VAR_INPUT
	id: INT;
END_VAR
CASE ID OF 
	1: 		GetMBMUData.s_Name:= 'Status';
			GetMBMUData.s_Type:= 'status';
			GetMBMUData.s_unit:= TO_STRING(data.e_BMS_Status);
	2: 		GetMBMUData.s_Name:= 'Power-on status';
			GetMBMUData.s_Type:= 'status';
			GetMBMUData.s_unit:= TO_STRING(data.e_BMS_PowerOnStatus);
	3:		GetMBMUData.s_Name:= 'Voltage';
			GetMBMUData.s_Type:= 'power';
			GetMBMUData.s_Unit:= 'VDC';
			GetMBMUData.i_precision:= 1;
			GetMBMUData.r_Data:= data.r_SystemVoltage;
	4:		GetMBMUData.s_Name:= 'Current';
			GetMBMUData.s_Type:= 'power';
			GetMBMUData.s_Unit:= 'A';
			GetMBMUData.i_precision:= 1;
			GetMBMUData.r_Data:= data.r_SystemCurrent;
	5:		GetMBMUData.s_Name:= 'Power';
			GetMBMUData.s_Type:= 'power';
			GetMBMUData.s_Unit:= 'kW';
			GetMBMUData.i_precision:= 1;
			GetMBMUData.r_Data:= data.r_SystemPower;
	6:		GetMBMUData.s_Name:= 'Max charge current';
			GetMBMUData.s_Type:= 'limit';
			GetMBMUData.s_Unit:= 'A';
			GetMBMUData.i_precision:= 1;
			GetMBMUData.r_Data:= data.r_MaxChargeCurrentAllowed;
	7:		GetMBMUData.s_Name:= 'Max discharge current';
			GetMBMUData.s_Type:= 'limit';
			GetMBMUData.s_Unit:= 'A';
			GetMBMUData.i_precision:= 1;
			GetMBMUData.r_Data:= data.r_MaxDischargeCurrentAllowed;
	8:		GetMBMUData.s_Name:= 'Max charge power';
			GetMBMUData.s_Type:= 'limit';
			GetMBMUData.s_Unit:= 'kW';
			GetMBMUData.i_precision:= 1;
			GetMBMUData.r_Data:= data.r_MaxChargePowerAllowed;
	9: 		GetMBMUData.s_Name:= 'Max discharge power';
			GetMBMUData.s_Type:= 'limit';
			GetMBMUData.s_Unit:= 'kW';
			GetMBMUData.i_precision:= 1;
			GetMBMUData.r_Data:= data.r_MaxDischargePowerAllowed;
	10:		GetMBMUData.s_Name:= 'Charge SOE';
			GetMBMUData.s_Type:= 'energy';
			GetMBMUData.s_Unit:= '%';
			GetMBMUData.i_precision:= 0;
			GetMBMUData.r_Data:= data.r_ChargeSOE;
	11:		GetMBMUData.s_Name:= 'Discharge SOE';                       
			GetMBMUData.s_Type:= 'energy';                       
			GetMBMUData.s_Unit:= '%';                               
			GetMBMUData.i_precision:= 0;                              
			GetMBMUData.r_Data:= data.r_DischargeSOE;
//	12:		GetMBMUData.s_Name:= 'Total charge energy';                       
//			GetMBMUData.s_Type:= 'energy';                       
//			GetMBMUData.s_Unit:= 'kWh';                               
//			GetMBMUData.i_precision:= 0;                              
//			GetMBMUData.r_Data:= data.r_HistAccChargeEnergy;
//	13:		GetMBMUData.s_Name:= 'Total discharge energy';                         
//			GetMBMUData.s_Type:= 'energy';                                 
//			GetMBMUData.s_Unit:= 'kWh';                                         
//			GetMBMUData.i_precision:= 0;                                        
//			GetMBMUData.r_Data:= data.r_HistAccDischargeEnergy;
			
	14:		GetMBMUData.s_Name:= 'Remaining charge energy';                         
			GetMBMUData.s_Type:= 'energy';                                 
			GetMBMUData.s_Unit:= 'kWh';                                         
			GetMBMUData.i_precision:= 0;                                        
			GetMBMUData.r_Data:= data.r_RemainingChargeEnergy;
	15:		GetMBMUData.s_Name:= 'Remaining discharge energy';                         
			GetMBMUData.s_Type:= 'energy';                                 
			GetMBMUData.s_Unit:= 'kWh';                                         
			GetMBMUData.i_precision:= 0;                                        
			GetMBMUData.r_Data:= data.r_RemainingDischargeEnergy;	
	16:		GetMBMUData.s_Name:= 'Max allowed voltage';                         
			GetMBMUData.s_Type:= 'limit';                                 
			GetMBMUData.s_Unit:= 'VDC';                                         
			GetMBMUData.i_precision:= 1;                                        
			GetMBMUData.r_Data:= data.r_MaxSystemVoltageAllowed;	
	17:		GetMBMUData.s_Name:= 'Min allowed voltage';                                     
			GetMBMUData.s_Type:= 'limit';                                     
			GetMBMUData.s_Unit:= 'VDC';                                             
			GetMBMUData.i_precision:= 1;                                            
			GetMBMUData.r_Data:= data.r_MinSystemVoltageAllowed;
			GetMBMUData.s_Type:= 'cell';                                        
			GetMBMUData.s_Unit:= 'VDC';                                                
			GetMBMUData.i_precision:= 2;                                               
			GetMBMUData.r_Data:= data.ar_CellVoltage[2];
	18:		GetMBMUData.s_Name:= 'SOH';
			GetMBMUData.s_Type:= 'status';
			GetMBMUData.s_Unit:= '%';
			GetMBMUData.i_precision:= 1;
			GetMBMUData.r_Data:= data.r_SOH;	
	19:		GetMBMUData.s_Name:= 'SOC actual';                          
			GetMBMUData.s_Type:= 'status';                  
			GetMBMUData.s_Unit:= '%';                            
			GetMBMUData.i_precision:= 1;                         
			GetMBMUData.r_Data:= data.r_SOC;
	20:		GetMBMUData.s_Name:= 'Cycle count';                          
			GetMBMUData.s_Type:= 'status';                                          
			GetMBMUData.s_unit:= TO_STRING(data.ui_CycleCount);
	ELSE	
		RETURN;			
END_CASE
END_METHOD

METHOD GetPowerModuleArrayData : ST_HMI_Monitor_ArrayDataFormat
VAR_IN_OUT CONSTANT
	data		: ST_Powermodule_get;
END_VAR

VAR_INPUT
	id: INT;
END_VAR
CASE ID OF 
	1: 		GetPowerModuleArrayData.s_Name:= 'Status';                                                
			GetPowerModuleArrayData.s_Type:= 'Status';                                                
			GetPowerModuleArrayData.s_Unit:= TO_STRING(data.e_Status);				                            
	2: 		GetPowerModuleArrayData.s_Name:= 'Inverter Mode';                                         
			GetPowerModuleArrayData.s_Type:= 'Status';                                                
			GetPowerModuleArrayData.s_Unit:= TO_STRING(data.e_InverterMode);					                     
	3:		GetPowerModuleArrayData.s_Name:= 'Power Mode';                                            
			GetPowerModuleArrayData.s_Type:= 'Status';                                                
			GetPowerModuleArrayData.s_Unit:= TO_STRING(data.e_PowerMode);						                       
	4:		GetPowerModuleArrayData.s_Name:= 'Fan state';                                             
			GetPowerModuleArrayData.s_Type:= 'Status';                                                
			GetPowerModuleArrayData.s_Unit:= SEL(data.b_FanFb,'OFF', 'RUNNING');						                
	5:		GetPowerModuleArrayData.s_Name:= 'MCCB state';                                            
			GetPowerModuleArrayData.s_Type:= 'Status';                                                
			GetPowerModuleArrayData.s_Unit:= SEL(data.b_MccbFb,'OPEN', 'CLOSED');						               
	6:		GetPowerModuleArrayData.s_Name:= 'MCCB tripstate';                                        
			GetPowerModuleArrayData.s_Type:= 'Status';                                                
			GetPowerModuleArrayData.s_Unit:= SEL(data.b_MccbTripOK,'TRIPPED', 'OK');						              
	7:		GetPowerModuleArrayData.s_Name:= 'D7 measurements OK';                                    
			GetPowerModuleArrayData.s_Type:= 'Ugrid statusword';                                      
			GetPowerModuleArrayData.s_Unit:= TO_STRING(data.UgridStatusWord.b_D7MeasurementsOK);						
	8:		GetPowerModuleArrayData.s_Name:= 'Synchronized to D7';                                    
			GetPowerModuleArrayData.s_Type:= 'Ugrid statusword';                                      
			GetPowerModuleArrayData.s_Unit:= TO_STRING(data.UgridStatusWord.b_SynchronizedToD7);      
	9: 		GetPowerModuleArrayData.s_Name:= 'Ready to DCcharge';                                     
			GetPowerModuleArrayData.s_Type:= 'statusword';                                            
			GetPowerModuleArrayData.s_Unit:= TO_STRING(data.StatusWord.b_ReadyToDCCharge);            
	10:		GetPowerModuleArrayData.s_Name:= 'Ready to operate';                                      
			GetPowerModuleArrayData.s_Type:= 'statusword';                                            
			GetPowerModuleArrayData.s_Unit:= TO_STRING(data.StatusWord.b_ReadyToOperate);
	11:		GetPowerModuleArrayData.s_Name:= 'Run enabled';                                           
			GetPowerModuleArrayData.s_Type:= 'statusword';                                            
			GetPowerModuleArrayData.s_Unit:= TO_STRING(data.StatusWord.b_RunEnabled);                 
	12:		GetPowerModuleArrayData.s_Name:= 'Running';                                               
			GetPowerModuleArrayData.s_Type:= 'statusword';                                            
			GetPowerModuleArrayData.s_Unit:= TO_STRING(data.StatusWord.b_Running);                    
	13:		GetPowerModuleArrayData.s_Name:= 'DC at reference';                                       
			GetPowerModuleArrayData.s_Type:= 'statusword';                                            
			GetPowerModuleArrayData.s_Unit:= TO_STRING(data.StatusWord.b_DCAtReference);              
	14:		GetPowerModuleArrayData.s_Name:= 'DC above limit';                                        
			GetPowerModuleArrayData.s_Type:= 'statusword';                                            
			GetPowerModuleArrayData.s_Unit:= TO_STRING(data.StatusWord.b_DCAboveLimit);               
	15:		GetPowerModuleArrayData.s_Name:= 'Quickstop active';                                      
			GetPowerModuleArrayData.s_Type:= 'statusword';                                            
			GetPowerModuleArrayData.s_Unit:= TO_STRING(NOT(data.StatusWord.b_QuickstopNotActive));    
	16:		GetPowerModuleArrayData.s_Name:= 'Warning';                                               
			GetPowerModuleArrayData.s_Type:= 'statusword';                                            
			GetPowerModuleArrayData.s_Unit:= TO_STRING(data.StatusWord.b_Warning);                    
	17:		GetPowerModuleArrayData.s_Name:= 'Fault';                                                 
			GetPowerModuleArrayData.s_Type:= 'statusword';                                            
			GetPowerModuleArrayData.s_Unit:= TO_STRING(data.StatusWord.b_Fault);                      
	18:		GetPowerModuleArrayData.s_Name:= 'MCCB control OK';                                       
			GetPowerModuleArrayData.s_Type:= 'statusword';                                            
			GetPowerModuleArrayData.s_Unit:= TO_STRING(NOT(data.StatusWord.b_MCCBControlNotOK));						
	19:		GetPowerModuleArrayData.s_Name:= 'Load';                                                   
			GetPowerModuleArrayData.s_Type:= 'AC';                                                    
			GetPowerModuleArrayData.s_Unit:= '%';                                                     
			GetPowerModuleArrayData.r_Data:= data.r_LoadPercent;                                      
			GetPowerModuleArrayData.i_precision := 1;	                                                
	20:		GetPowerModuleArrayData.s_Name:= 'Apparent Power';                                        
			GetPowerModuleArrayData.s_Type:= 'AC';                                                    
			GetPowerModuleArrayData.s_Unit:= 'kVA';                                                   
			GetPowerModuleArrayData.r_Data:= data.r_ApparentPower;                                    
			GetPowerModuleArrayData.i_precision := 0;                                                 
	21:		GetPowerModuleArrayData.s_Name:= 'Active Power';                                          
			GetPowerModuleArrayData.s_Type:= 'AC';                                                    
			GetPowerModuleArrayData.s_Unit:= 'kW';                                                    
			GetPowerModuleArrayData.r_Data:= data.r_ActivePower;                                      
			GetPowerModuleArrayData.i_precision := 1;                                                 
	22:		GetPowerModuleArrayData.s_Name:= 'Reactive Power';                                        
			GetPowerModuleArrayData.s_Type:= 'AC';                                                    
			GetPowerModuleArrayData.s_Unit:= 'kvar';                                                  
			GetPowerModuleArrayData.r_Data:= data.r_ReactivePower;                                    
			GetPowerModuleArrayData.i_precision := 1;                                                 
	23:		GetPowerModuleArrayData.s_Name:= 'Current';                                               
			GetPowerModuleArrayData.s_Type:= 'AC';                                                    
			GetPowerModuleArrayData.s_Unit:= 'A';                                                     
			GetPowerModuleArrayData.r_Data:= data.r_ACCurrent;                                        
			GetPowerModuleArrayData.i_precision := 1;                                                 
	24:		GetPowerModuleArrayData.s_Name:= 'Reactive Current';                                      
			GetPowerModuleArrayData.s_Type:= 'AC';                                                    
			GetPowerModuleArrayData.s_Unit:= 'A';                                                     
			GetPowerModuleArrayData.r_Data:= data.r_ReactiveCurrent;                                  
			GetPowerModuleArrayData.i_precision := 1;                                                 
	25:		GetPowerModuleArrayData.s_Name:= 'Active Current';                                        
			GetPowerModuleArrayData.s_Type:= 'AC';                                                    
			GetPowerModuleArrayData.s_Unit:= 'A';                                                     
			GetPowerModuleArrayData.r_Data:= data.r_ActiveCurrent;                                    
			GetPowerModuleArrayData.i_precision := 1;                                                 
	26:		GetPowerModuleArrayData.s_Name:= 'Supply Voltage';                                        
			GetPowerModuleArrayData.s_Type:= 'AC';                                                    
			GetPowerModuleArrayData.s_Unit:= 'VAC';                                                   
			GetPowerModuleArrayData.r_Data:= data.r_ACVoltageSupply;                                  
			GetPowerModuleArrayData.i_precision := 1;                                                 
	27:		GetPowerModuleArrayData.s_Name:= 'Supply Frequency';                                      
			GetPowerModuleArrayData.s_Type:= 'AC';                                                    
			GetPowerModuleArrayData.s_Unit:= 'Hz';                                                    
			GetPowerModuleArrayData.r_Data:= data.r_FrequencySupply;                                  
			GetPowerModuleArrayData.i_precision := 2;                                                 
	28:		GetPowerModuleArrayData.s_Name:= 'Current';                                               
			GetPowerModuleArrayData.s_Type:= 'DC';                                                    
			GetPowerModuleArrayData.s_Unit:= 'A';                                                     
			GetPowerModuleArrayData.r_Data:= data.r_DCCurrent;                                        
			GetPowerModuleArrayData.i_precision := 1;                                                 
	29:		GetPowerModuleArrayData.s_Name:= 'Voltage';                                               
			GetPowerModuleArrayData.s_Type:= 'DC';                                                    
			GetPowerModuleArrayData.s_Unit:= 'VDC';                                                   
			GetPowerModuleArrayData.r_Data:= data.r_DCVoltage;                                        
			GetPowerModuleArrayData.i_precision := 1;                                                 
	30:		GetPowerModuleArrayData.s_Name:= 'Power';                                                 
			GetPowerModuleArrayData.s_Type:= 'DC';                                                    
			GetPowerModuleArrayData.s_Unit:= 'kW';                                                    
			GetPowerModuleArrayData.r_Data:= data.r_DCPower;                                          
			GetPowerModuleArrayData.i_precision := 1;                                                 
	31:		GetPowerModuleArrayData.s_Name:= 'CMchoke L1';                                            
			GetPowerModuleArrayData.s_Type:= 'Temperatures';                                          
			GetPowerModuleArrayData.s_Unit:= '°C';                                                    
			GetPowerModuleArrayData.r_Data:= data.r_TemperatureCMChoke[1];                            
			GetPowerModuleArrayData.i_precision := 1;                                                 
	32:		GetPowerModuleArrayData.s_Name:= 'CMchoke L2';                                            
			GetPowerModuleArrayData.s_Type:= 'Temperatures';                                          
			GetPowerModuleArrayData.s_Unit:= '°C';                                                    
			GetPowerModuleArrayData.r_Data:= data.r_TemperatureCMChoke[2];                            
			GetPowerModuleArrayData.i_precision := 1;                                                 
	33:		GetPowerModuleArrayData.s_Name:= 'CMchoke L3';                                            
			GetPowerModuleArrayData.s_Type:= 'Temperatures';                                          
			GetPowerModuleArrayData.s_Unit:= '°C';                                                    
			GetPowerModuleArrayData.r_Data:= data.r_TemperatureCMChoke[3];                            
			GetPowerModuleArrayData.i_precision := 1;                                                 
	34:		GetPowerModuleArrayData.s_Name:= 'CMchoke DC';                                            
			GetPowerModuleArrayData.s_Type:= 'Temperatures';                                          
			GetPowerModuleArrayData.s_Unit:= '°C';                                                    
			GetPowerModuleArrayData.r_Data:= data.r_TemperatureCMChoke[4];                            
			GetPowerModuleArrayData.i_precision := 1;                                                 
	35:		GetPowerModuleArrayData.s_Name:= 'Gridchoke L1';                                          
			GetPowerModuleArrayData.s_Type:= 'Temperatures';                                          
			GetPowerModuleArrayData.s_Unit:= '°C';                                                    
			GetPowerModuleArrayData.r_Data:= data.r_Temperaturegridchoke[1];                          
			GetPowerModuleArrayData.i_precision := 1;                                                 
	36:		GetPowerModuleArrayData.s_Name:= 'Gridchoke L2';                                          
			GetPowerModuleArrayData.s_Type:= 'Temperatures';                                          
			GetPowerModuleArrayData.s_Unit:= '°C';                                                    
			GetPowerModuleArrayData.r_Data:= data.r_Temperaturegridchoke[2];                          
			GetPowerModuleArrayData.i_precision := 1;                                                 
	37:		GetPowerModuleArrayData.s_Name:= 'Gridchoke L3';                                          
			GetPowerModuleArrayData.s_Type:= 'Temperatures';                                          
			GetPowerModuleArrayData.s_Unit:= '°C';                                                    
			GetPowerModuleArrayData.r_Data:= data.r_Temperaturegridchoke[3];                          
			GetPowerModuleArrayData.i_precision := 1;                                                 
	38:		GetPowerModuleArrayData.s_Name:= 'Inverter';                                              
			GetPowerModuleArrayData.s_Type:= 'Temperatures';                                          
			GetPowerModuleArrayData.s_Unit:= '°C';                                                    
			GetPowerModuleArrayData.r_Data:= data.r_TemperatureInverter;                              
			GetPowerModuleArrayData.i_precision := 1;                                                 
	39:		GetPowerModuleArrayData.s_Name:= 'Powermodule max';                                   
			GetPowerModuleArrayData.s_Type:= 'Temperatures';                                          
			GetPowerModuleArrayData.s_Unit:= '°C';                                                    
			GetPowerModuleArrayData.r_Data:= data.r_TemperatureMax;                                   
			GetPowerModuleArrayData.i_precision := 1;                                                 
	40:		GetPowerModuleArrayData.s_Name:= 'Active power min(charge)';                              
			GetPowerModuleArrayData.s_Type:= 'Limits';                                                
			GetPowerModuleArrayData.s_Unit:= 'kW';                                                    
			GetPowerModuleArrayData.r_Data:= data.r_Pmin;                                             
			GetPowerModuleArrayData.i_precision := 0;                                                 
	41:		GetPowerModuleArrayData.s_Name:= 'Active power max (discharge)';                          
			GetPowerModuleArrayData.s_Type:= 'Limits';                                                
			GetPowerModuleArrayData.s_Unit:= 'kW';                                                    
			GetPowerModuleArrayData.r_Data:= data.r_Pmax;                                             
			GetPowerModuleArrayData.i_precision := 0;                                                 
	42:		GetPowerModuleArrayData.s_Name:= 'Reactive power min';                                    
			GetPowerModuleArrayData.s_Type:= 'Limits';                                                
			GetPowerModuleArrayData.s_Unit:= 'kvar';                                                  
			GetPowerModuleArrayData.r_Data:= data.r_QMin;                                             
			GetPowerModuleArrayData.i_precision := 0;                                                 
	43:		GetPowerModuleArrayData.s_Name:= 'Reactive power max';                                    
			GetPowerModuleArrayData.s_Type:= 'Limits';                                                
			GetPowerModuleArrayData.s_Unit:= 'kvar';                                                  
			GetPowerModuleArrayData.r_Data:= data.r_QMax;                                             
			GetPowerModuleArrayData.i_precision := 0;                                                 
	44:		GetPowerModuleArrayData.s_Name:= 'D7 Sync Error';                                         
			GetPowerModuleArrayData.s_Type:= 'AC';                                           
			GetPowerModuleArrayData.s_Unit:= '°';                                                     
			GetPowerModuleArrayData.r_Data:= data.r_D7SyncError;                                      
			GetPowerModuleArrayData.i_precision := 1;
	45:		GetPowerModuleArrayData.s_Name:= 'Active power';                                         
			GetPowerModuleArrayData.s_Type:= 'Setpoints';                                           
			GetPowerModuleArrayData.s_Unit:= 'kW';                                                     
			GetPowerModuleArrayData.r_Data:= data.r_Pset;                                      
			GetPowerModuleArrayData.i_precision := 0; 
	46:		GetPowerModuleArrayData.s_Name:= 'Reactive power';                                         
			GetPowerModuleArrayData.s_Type:= 'Setpoints';                                           
			GetPowerModuleArrayData.s_Unit:= 'kvar';                                                     
			GetPowerModuleArrayData.r_Data:= data.r_Qset;                                      
			GetPowerModuleArrayData.i_precision := 1;   
	47:		GetPowerModuleArrayData.s_Name:= 'Base current ref';                                         
			GetPowerModuleArrayData.s_Type:= 'Controls';                                           
			GetPowerModuleArrayData.s_Unit:= '0.1%';                                                     
			GetPowerModuleArrayData.r_Data:= data.ControlData.i_BaseCurrentRef;                                      
			GetPowerModuleArrayData.i_precision := 0; 
	48:		GetPowerModuleArrayData.s_Name:= 'Reactive current ref';                                         
			GetPowerModuleArrayData.s_Type:= 'Controls';                                           
			GetPowerModuleArrayData.s_Unit:= '0.1%';                                                     
			GetPowerModuleArrayData.r_Data:= data.ControlData.i_ReactiveCurrentRef;                                      
			GetPowerModuleArrayData.i_precision := 0;
	49:		GetPowerModuleArrayData.s_Name:= 'Frequency droop offset';                                         
			GetPowerModuleArrayData.s_Type:= 'Controls';                                           
			GetPowerModuleArrayData.s_Unit:= '0.1Hz';                                                     
			GetPowerModuleArrayData.r_Data:= data.ControlData.i_FrequencyDroopOffset;                                      
			GetPowerModuleArrayData.i_precision := 0;
	50:		GetPowerModuleArrayData.s_Name:= 'Voltage correction';                                         
			GetPowerModuleArrayData.s_Type:= 'Controls';                                           
			GetPowerModuleArrayData.s_Unit:= 'V';                                                     
			GetPowerModuleArrayData.r_Data:= data.ControlData.i_VoltageCorrection;
            GetPowerModuleArrayData.i_precision := 0;
	51:		GetPowerModuleArrayData.s_Name:= 'Frequency Droop';                                         
			GetPowerModuleArrayData.s_Type:= 'Controls';                                           
			GetPowerModuleArrayData.s_Unit:= '0.001Hz';                                                     
			GetPowerModuleArrayData.r_Data:= data.ControlData.i_FrequencyDroop;
            GetPowerModuleArrayData.i_precision := 0;  
	52:		GetPowerModuleArrayData.s_Name:= 'Voltage Droop';                                         
			GetPowerModuleArrayData.s_Type:= 'Controls';                                           
			GetPowerModuleArrayData.s_Unit:= '0.01%';                                                     
			GetPowerModuleArrayData.r_Data:= data.ControlData.i_VoltageDroop;
            GetPowerModuleArrayData.i_precision := 0;  
	53:		GetPowerModuleArrayData.s_Name:= 'Base ref ramprate';                                         
			GetPowerModuleArrayData.s_Type:= 'Controls';                                           
			GetPowerModuleArrayData.s_Unit:= '%';                                                     
			GetPowerModuleArrayData.r_Data:= data.ControlData.i_BaseRefRampRate;
            GetPowerModuleArrayData.i_precision := 0;  
    54:		GetPowerModuleArrayData.s_Name:= 'Start Powermode';                                         
			GetPowerModuleArrayData.s_Type:= 'Controls';                                           
			GetPowerModuleArrayData.s_Unit:= '-';                                                     
			GetPowerModuleArrayData.r_Data:= data.ControlData.i_StartPowerMode;
            GetPowerModuleArrayData.i_precision := 0;
    55:		GetPowerModuleArrayData.s_Name:= 'Start Voltagemode';                                         
			GetPowerModuleArrayData.s_Type:= 'Controls';                                           
			GetPowerModuleArrayData.s_Unit:= '%';                                                     
			GetPowerModuleArrayData.r_Data:= data.ControlData.i_StartVoltageMode;
            GetPowerModuleArrayData.i_precision := 0; 
	56:		GetPowerModuleArrayData.s_Name:= 'Output act. current limit';                                         
			GetPowerModuleArrayData.s_Type:= 'Controls';                                           
			GetPowerModuleArrayData.s_Unit:= '0.1%';                                                     
			GetPowerModuleArrayData.r_Data:= data.ControlData.i_OutActCurrentLimit;
            GetPowerModuleArrayData.i_precision := 0;
	57:		GetPowerModuleArrayData.s_Name:= 'Input act. current limit';                                         
			GetPowerModuleArrayData.s_Type:= 'Controls';                                           
			GetPowerModuleArrayData.s_Unit:= '0.1%';                                                     
			GetPowerModuleArrayData.r_Data:= data.ControlData.i_InActCurrentLimit;
            GetPowerModuleArrayData.i_precision := 0;                                                                                                            
	ELSE	
		RETURN;			
END_CASE
END_METHOD

METHOD	GetPowerstackArrayData : ST_HMI_Monitor_ArrayDataFormat

VAR_INPUT
	id: INT;
END_VAR
CASE ID OF 
	1: 		GetPowerstackArrayData.s_Name:= 'Status';                              
			GetPowerstackArrayData.s_Type:= 'Status';                              
			GetPowerstackArrayData.s_Unit:= TO_STRING(monitor.PowerStack.e_State);
	3:		GetPowerstackArrayData.s_Name:= 'Load';                              
			GetPowerstackArrayData.s_Type:= 'AC';                                
			GetPowerstackArrayData.s_Unit:= '%';                                 
			GetPowerstackArrayData.r_Data:= monitor.PowerStack.r_LoadPercent;    
			GetPowerstackArrayData.i_precision := 1;	                                             
	4:		GetPowerstackArrayData.s_Name:= 'Apparent Power';                    
			GetPowerstackArrayData.s_Type:= 'AC';                                
			GetPowerstackArrayData.s_Unit:= 'kVA';                               
			GetPowerstackArrayData.r_Data:= monitor.PowerStack.r_ApparentPower;  
			GetPowerstackArrayData. i_precision := 0;                                             
	5:		GetPowerstackArrayData.s_Name:= 'Active Power';                      
			GetPowerstackArrayData.s_Type:= 'AC';                                
			GetPowerstackArrayData.s_Unit:= 'kW';                                
			GetPowerstackArrayData.r_Data:= monitor.PowerStack.r_ActivePower;    
			GetPowerstackArrayData.i_precision := 1;                                             
	6:		GetPowerstackArrayData.s_Name:= 'Reactive Power';                    
			GetPowerstackArrayData.s_Type:= 'AC';                                
			GetPowerstackArrayData.s_Unit:= 'kvar';                              
			GetPowerstackArrayData.r_Data:= monitor.PowerStack.r_ReactivePower;  
			GetPowerstackArrayData.i_precision := 1;                                             
	7:		GetPowerstackArrayData.s_Name:= 'Current';                           
			GetPowerstackArrayData.s_Type:= 'AC';                                
			GetPowerstackArrayData.s_Unit:= 'A';                                 
			GetPowerstackArrayData.r_Data:= monitor.PowerStack.r_ACCurrent;      
			GetPowerstackArrayData.i_precision := 1;                                              
	8:		GetPowerstackArrayData.s_Name:= 'Supply Voltage';                    
			GetPowerstackArrayData.s_Type:= 'AC';                                
			GetPowerstackArrayData.s_Unit:= 'VAC';                               
			GetPowerstackArrayData.r_Data:= monitor.PowerStack.r_ACVoltageSupply;
			GetPowerstackArrayData.i_precision := 1;                                              
	9: 		GetPowerstackArrayData.s_Name:= 'Supply Frequency';                  
			GetPowerstackArrayData.s_Type:= 'AC';                                
			GetPowerstackArrayData.s_Unit:= 'Hz';                                
			GetPowerstackArrayData.r_Data:= monitor.PowerStack.r_FrequencySupply;
			GetPowerstackArrayData.i_precision := 2;
	10:		GetPowerstackArrayData.s_Name:= 'D7 Voltage';                    
			GetPowerstackArrayData.s_Type:= 'AC';                                
			GetPowerstackArrayData.s_Unit:= 'VAC';                               
			GetPowerstackArrayData.r_Data:= monitor.PowerStack.r_ACVoltageD7;
			GetPowerstackArrayData.i_precision := 0;                                              
	11: 	GetPowerstackArrayData.s_Name:= 'D7 Frequency';                  
			GetPowerstackArrayData.s_Type:= 'AC';                                
			GetPowerstackArrayData.s_Unit:= 'Hz';                                
			GetPowerstackArrayData.r_Data:= monitor.PowerStack.r_FrequencyD7;
			GetPowerstackArrayData.i_precision := 2;                                                                                    
	12:		GetPowerstackArrayData.s_Name:= 'Cos Phi';                           
			GetPowerstackArrayData.s_Type:= 'AC';                                
			GetPowerstackArrayData.s_Unit:= '-';                                 
			GetPowerstackArrayData.r_Data:= monitor.PowerStack.r_Cosphi;         
			GetPowerstackArrayData.i_precision := 2;
	13:		GetPowerstackArrayData.s_Name:= 'Current';                           
			GetPowerstackArrayData.s_Type:= 'DC';                                
			GetPowerstackArrayData.s_Unit:= 'A';                                 
			GetPowerstackArrayData.r_Data:= monitor.PowerStack.r_DCCurrent;      
			GetPowerstackArrayData.i_precision := 1;                                              
	14:		GetPowerstackArrayData.s_Name:= 'Voltage';                           
			GetPowerstackArrayData.s_Type:= 'DC';                                
			GetPowerstackArrayData.s_Unit:= 'VDC';                               
			GetPowerstackArrayData.r_Data:= monitor.PowerStack.r_DCVoltage;      
			GetPowerstackArrayData.i_precision := 1;                                              
	15:		GetPowerstackArrayData.s_Name:= 'Power';                             
			GetPowerstackArrayData.s_Type:= 'DC';                                
			GetPowerstackArrayData.s_Unit:= 'kW';                                
			GetPowerstackArrayData.r_Data:= monitor.PowerStack.r_DCPower; 
			GetPowerstackArrayData.i_precision := 1;        
	16:		GetPowerstackArrayData.s_Name:= 'Inverter Mode';                                         
			GetPowerstackArrayData.s_Type:= 'Status';                                                
			GetPowerstackArrayData.s_Unit:= TO_STRING(monitor.PowerStack.e_InverterMode);            
	17:		GetPowerstackArrayData.s_Name:= 'Power Mode';                                            
			GetPowerstackArrayData.s_Type:= 'Status';                                                
			GetPowerstackArrayData.s_Unit:= TO_STRING(monitor.PowerStack.e_PowerMode);               
	18:		GetPowerstackArrayData.s_Name:= 'Netcontactor';                                          
			GetPowerstackArrayData.s_Type:= 'Status';                                                
			GetPowerstackArrayData.s_Unit:= TO_STRING(monitor.PowerStack.NetContactor.e_NetConState);
	19: 	GetPowerstackArrayData.s_Name:= 'Energy out';      
			GetPowerstackArrayData.s_Type:= 'Energy';         
			GetPowerstackArrayData.s_Unit:= 'kWh';            
			GetPowerstackArrayData.i_precision:= 1;
			GetPowerstackArrayData.b_warning := monitor.powermonitor.BESS.r_EnergySupplied < 0;              
			GetPowerstackArrayData.r_Data:= monitor.powermonitor.BESS.r_EnergySupplied;
	20: 	GetPowerstackArrayData.s_Name:= 'Energy in';          
			GetPowerstackArrayData.s_Type:= 'Energy';         
			GetPowerstackArrayData.s_Unit:= 'kWh';                
			GetPowerstackArrayData.i_precision:= 1;
			GetPowerstackArrayData.b_warning := monitor.powermonitor.BESS.r_EnergyConsumed < 0;              
			GetPowerstackArrayData.r_Data:= monitor.powermonitor.BESS.r_EnergyConsumed;
	ELSE	
		RETURN;
END_CASE
END_METHOD

METHOD	GetPSBdata : ST_HMI_Monitor_ArrayDataFormat
VAR_IN_OUT CONSTANT
	data : ST_Peakshavebox_get;
END_VAR

VAR_INPUT
	id: INT;
END_VAR
CASE ID OF 
	1: 		GetPSBData.s_Name:= 'Breaker state';
			GetPSBData.s_Type:= 'Status';
			GetPSBData.s_Unit:= SEL(data.b_ContactorFb, 'OPEN', 'CLOSED');
	2: 		GetPSBData.s_Name:= 'Sync state';
			GetPSBData.s_Type:= 'Status';
			GetPSBData.s_Unit:= TO_STRING(data.b_SyncFb);
	3:		GetPSBData.s_Name:= 'Apparent Power';
			GetPSBData.s_Type:= 'AC';
			GetPSBData.s_Unit:= 'kVA';
			GetPSBData.i_precision:= 0;
			GetPSBData.r_Data:= data.Powermonitor.ar_ApparentPower[0];
	4:		GetPSBData.s_Name:= 'Active Power';
			GetPSBData.s_Type:= 'AC';
			GetPSBData.s_Unit:= 'kW';
			GetPSBData.i_precision:= 1;
			GetPSBData.r_Data:= data.Powermonitor.ar_ActivePower[0];
	5:		GetPSBData.s_Name:= 'Reactive Power';
			GetPSBData.s_Type:= 'AC';
			GetPSBData.s_Unit:= 'kvar';
			GetPSBData.i_precision:= 1;
			GetPSBData.r_Data:= data.Powermonitor.ar_ReactivePower[0];
	6:		GetPSBData.s_Name:= 'Current';
			GetPSBData.s_Type:= 'AC';
			GetPSBData.s_Unit:= 'A';
			GetPSBData.i_precision:= 1;
			GetPSBData.r_Data:= data.Powermonitor.ar_Current[0];
	7:		GetPSBData.s_Name:= 'Line Voltage';
			GetPSBData.s_Type:= 'AC';
			GetPSBData.s_Unit:= 'VAC';
			GetPSBData.i_precision:= 1;
			GetPSBData.r_Data:= data.powermonitor.ar_LineVoltage[0];
	8:		GetPSBData.s_Name:= 'Phase Voltage';
			GetPSBData.s_Type:= 'AC';
			GetPSBData.s_Unit:= 'VAC';
			GetPSBData.i_precision:= 1;
			GetPSBData.r_Data:= data.powermonitor.ar_PhaseVoltage[0];
	9:		GetPSBData.s_Name:= 'Frequency';
			GetPSBData.s_Type:= 'AC';
			GetPSBData.s_Unit:= 'Hz';
			GetPSBData.i_precision:= 2;
			GetPSBData.r_Data:=  data.powermonitor.ar_Frequency[0];
	10: 	GetPSBData.s_Name:= 'Power factor';
			GetPSBData.s_Type:= 'AC';
			GetPSBData.s_Unit:= '-';
			GetPSBData.i_precision:= 2;
			GetPSBData.r_Data:=  data.powermonitor.ar_Powerfactor[0];
	11:		GetPSBData.s_Name:= 'L1';
			GetPSBData.s_Type:= 'AC Current';
			GetPSBData.s_Unit:= 'A';
			GetPSBData.i_precision:= 1;
			GetPSBData.r_Data:= data.Powermonitor.ar_Current[1];
	12:		GetPSBData.s_Name:= 'L2';
			GetPSBData.s_Type:= 'AC Current';
			GetPSBData.s_Unit:= 'A';
			GetPSBData.i_precision:= 1;
			GetPSBData.r_Data:= data.Powermonitor.ar_Current[2];
	13:		GetPSBData.s_Name:= 'L3';
			GetPSBData.s_Type:= 'AC Current';
			GetPSBData.s_Unit:= 'A';
			GetPSBData.i_precision:= 1;
			GetPSBData.r_Data:= data.Powermonitor.ar_Current[3];
	15:		GetPSBData.s_Name:= 'N';
			GetPSBData.s_Type:= 'AC Current';
			GetPSBData.s_Unit:= 'A';
			GetPSBData.i_precision:= 1;
			GetPSBData.r_Data:= data.Powermonitor.ar_Current[4];	
	16:		GetPSBData.s_Name:= 'L1-L2';
			GetPSBData.s_Type:= 'AC Linevoltage';
			GetPSBData.s_Unit:= 'VAC';
			GetPSBData.i_precision:= 1;
			GetPSBData.r_Data:= data.powermonitor.ar_LineVoltage[1];
	17:		GetPSBData.s_Name:= 'L2-L3';
			GetPSBData.s_Type:= 'AC Linevoltage';
			GetPSBData.s_Unit:= 'VAC';
			GetPSBData.i_precision:= 1;
			GetPSBData.r_Data:= data.powermonitor.ar_LineVoltage[2];
	18:		GetPSBData.s_Name:= 'L3-L1';
			GetPSBData.s_Type:= 'AC Linevoltage';
			GetPSBData.s_Unit:= 'VAC';
			GetPSBData.i_precision:= 1;
			GetPSBData.r_Data:= data.powermonitor.ar_LineVoltage[3];
	19:		GetPSBData.s_Name:= 'L1-N';
			GetPSBData.s_Type:= 'AC Phasevoltage';
			GetPSBData.s_Unit:= 'VAC';
			GetPSBData.i_precision:= 1;
			GetPSBData.r_Data:= data.powermonitor.ar_PhaseVoltage[1];
	20:		GetPSBData.s_Name:= 'L2-N';
			GetPSBData.s_Type:= 'AC Phasevoltage';
			GetPSBData.s_Unit:= 'VAC';
			GetPSBData.i_precision:= 1;
			GetPSBData.r_Data:= data.powermonitor.ar_PhaseVoltage[2];
	21:		GetPSBData.s_Name:= 'L3-N';
			GetPSBData.s_Type:= 'AC Phasevoltage';
			GetPSBData.s_Unit:= 'VAC';
			GetPSBData.i_precision:= 1;
			GetPSBData.r_Data:= data.powermonitor.ar_PhaseVoltage[3];					
	22:		GetPSBData.s_Name:= 'Rotation field';
			GetPSBData.s_Type:= 'AC';
			GetPSBData.s_Unit:= SEL(data.Powerstatus.b_RotaryField, 'RIGHT', 'LEFT');
	23: 	GetPSBData.s_Name:= 'Energy in';                 
			GetPSBData.s_Type:= 'Energy'; 
			GetPSBData.s_Unit:= 'kWh';                 
			GetPSBData.i_precision:= 0;
			GetPSBData.b_warning := monitor.powermonitor.outputfield.r_EnergyConsumed < 0;              
			GetPSBData.r_Data:= data.powermonitor.r_EnergyConsumed;
	24: 	GetPSBData.s_Name:= 'Energy out';                 
			GetPSBData.s_Type:= 'Energy'; 
			GetPSBData.s_Unit:= 'kWh';                 
			GetPSBData.i_precision:= 0;
			GetPSBData.b_warning := monitor.powermonitor.outputfield.r_EnergySupplied < 0;              
			GetPSBData.r_Data:= data.powermonitor.r_EnergySupplied;
ELSE	
		RETURN;
END_CASE
END_METHOD

METHOD GetSBMUData : ST_HMI_Monitor_ArrayDataFormat
VAR_IN_OUT CONSTANT
	data 			: st_SBMU_Status;
END_VAR

VAR_INPUT
	id: INT;
	SBMU_NO	: BYTE;
END_VAR
CASE ID OF 
	1: 		GetSBMUData.s_Name:= 'Warning word';
			GetSBMUData.s_Type:= 'status';
			GetSBMUData.s_unit:= TO_STRING(data.w_SystemWarning);
	2: 		GetSBMUData.s_Name:= 'Precharge Relay';
			GetSBMUData.s_Type:= 'status';
			GetSBMUData.s_unit:= SEL(data.b_PrechargeRelayClosed, 'OPEN', 'CLOSED');
	3: 		GetSBMUData.s_Name:= 'Positive Relay';
			GetSBMUData.s_Type:= 'status';
			GetSBMUData.s_unit:= SEL(data.b_MainPosRelayClosed,'OPEN', 'CLOSED');
	4: 		GetSBMUData.s_Name:= 'Negative Relay';
			GetSBMUData.s_Type:= 'status';
			GetSBMUData.s_unit:= SEL(data.b_MainNegRelayClosed,'OPEN', 'CLOSED');
	5: 		GetSBMUData.s_Name:= 'Fan';
			GetSBMUData.s_Type:= 'status';
			GetSBMUData.s_unit:= SEL(data.b_ControlBoxFanOn,'ON', 'OFF');
	6: 		GetSBMUData.s_Name:= 'Balance status';
			GetSBMUData.s_Type:= 'status';
			GetSBMUData.s_unit:= SEL(data.b_BalanceStatus,'ON', 'OFF');
	7:		GetSBMUData.s_Name:= 'Voltage';
			GetSBMUData.s_Type:= 'power';
			GetSBMUData.s_Unit:= 'VDC';
			GetSBMUData.i_precision:= 1;
			GetSBMUData.r_Data:= data.BatteryStatus.r_SystemVoltage;
	8:		GetSBMUData.s_Name:= 'Current';
			GetSBMUData.s_Type:= 'power';
			GetSBMUData.s_Unit:= 'A';
			GetSBMUData.i_precision:= 0;
			GetSBMUData.r_Data:= data.BatteryStatus.r_SystemCurrent;
	9:		GetSBMUData.s_Name:= 'Max charge current';
			GetSBMUData.s_Type:= 'limit';
			GetSBMUData.s_Unit:= 'A';
			GetSBMUData.i_precision:= 0;
			GetSBMUData.r_Data:= data.BatteryStatus.r_MaxChargeCurrentAllowed;
	10:		GetSBMUData.s_Name:= 'Max discharge current';
			GetSBMUData.s_Type:= 'limit';
			GetSBMUData.s_Unit:= 'A';
			GetSBMUData.i_precision:= 0;
			GetSBMUData.r_Data:= data.BatteryStatus.r_MaxDischargeCurrentAllowed;
	11:		GetSBMUData.s_Name:= 'Total charge energy';                       
			GetSBMUData.s_Type:= 'energy';                       
			GetSBMUData.s_Unit:= 'kWh';                               
			GetSBMUData.i_precision:= 0;                              
			GetSBMUData.r_Data:= data.BatteryStatus.r_HistAccChargeEnergy;
	12:		GetSBMUData.s_Name:= 'Total discharge energy';                         
			GetSBMUData.s_Type:= 'energy';                                 
			GetSBMUData.s_Unit:= 'kWh';                                         
			GetSBMUData.i_precision:= 0;                                        
			GetSBMUData.r_Data:= data.BatteryStatus.r_HistAccDischargeEnergy;
	13:		GetSBMUData.s_Name:= 'Min. cell temperature';                               
			GetSBMUData.s_Type:= 'cell';                                        
			GetSBMUData.s_Unit:= '°C';                                                
			GetSBMUData.i_precision:= 2;                                               
			GetSBMUData.r_Data:= data.BatteryStatus.ar_CellTemperature[0];
	14:		GetSBMUData.s_Name:= 'Avg. cell temperature';                               
			GetSBMUData.s_Type:= 'cell';                                        
			GetSBMUData.s_Unit:= '°C';                                                
			GetSBMUData.i_precision:= 2;                                               
			GetSBMUData.r_Data:= data.BatteryStatus.ar_CellTemperature[1];	
	15:		GetSBMUData.s_Name:= 'Max. cell temperature';                               
			GetSBMUData.s_Type:= 'cell';                                        
			GetSBMUData.s_Unit:= '°C';                                                
			GetSBMUData.i_precision:= 2;                                               
			GetSBMUData.r_Data:= data.BatteryStatus.ar_CellTemperature[2];
	16:		GetSBMUData.s_Name:= 'Min. cell voltage';                               
			GetSBMUData.s_Type:= 'cell';                                        
			GetSBMUData.s_Unit:= 'VDC';                                                
			GetSBMUData.i_precision:= 2;                                               
			GetSBMUData.r_Data:= monitor.battery.BatteryInfo.ar_Cellvoltage[0];
	17:		GetSBMUData.s_Name:= 'Avg. cell voltage';                               
			GetSBMUData.s_Type:= 'cell';                                        
			GetSBMUData.s_Unit:= 'VDC';                                                
			GetSBMUData.i_precision:= 2;                                               
			GetSBMUData.r_Data:= data.BatteryStatus.ar_CellVoltage[1];	
	18:		GetSBMUData.s_Name:= 'Max. cell voltage';                               
			GetSBMUData.s_Type:= 'cell';                                        
			GetSBMUData.s_Unit:= 'VDC';                                                
			GetSBMUData.i_precision:= 2;                                               
			GetSBMUData.r_Data:= data.BatteryStatus.ar_CellVoltage[2];
	19:		GetSBMUData.s_Name:= 'SOH';
			GetSBMUData.s_Type:= 'status';
			GetSBMUData.s_Unit:= '%';
			GetSBMUData.i_precision:= 1;
			GetSBMUData.r_Data:= data.BatteryStatus.r_SOH;	
	20:		GetSBMUData.s_Name:= 'SOC actual';                          
			GetSBMUData.s_Type:= 'status';                  
			GetSBMUData.s_Unit:= '%';                            
			GetSBMUData.i_precision:= 1;                         
			GetSBMUData.r_Data:= data.BatteryStatus.r_SOC;	
	21: 	GetSBMUData.s_Name:= 'ID';                          
			GetSBMUData.s_Type:= 'ID';                                                                    
			GetSBMUData.r_Data:= SBMU_NO;
	ELSE	
		RETURN;			
END_CASE
END_METHOD

METHOD PRIVATE Hour_Minute_To_TOW : WORD
VAR_INPUT
	dayofweek: USINT;
	hour	: USINT;
	minute	: USINT;
END_VAR
Hour_Minute_To_TOW := dayofweek * 24 * 60 + hour * 60 + minute;
END_METHOD

ACTION MapPLCvarsToHMIVars:
//System
	monitoringvars.System.e_SystemState 				:= monitor.system.e_State;
	monitoringvars.System.b_startAllowed				:= monitor.system.b_StartAllowed;
	monitoringvars.System.e_GridMode					:= monitor.system.e_gridmode;
	monitoringvars.System.e_UgridPowermode				:= monitor.system.e_UgridPowermode;
	monitoringvars.System.b_earthingSelected			:= monitor.controlfb.HardSettings.system.e_EarthingSystem <> eEarthingsystems.None;
	monitoringvars.System.b_CustomNameConfigured		:= monitor.system.b_CustomNameConfigured;
	monitoringvars.System.b_SMSnumberConfigured			:= monitor.system.b_SMSnumberConfigured;
	monitoringvars.System.r_averageEfficiency			:= monitor.system.r_AvgEfficiency;
	monitoringvars.System.r_currentEfficiency			:= monitor.system.r_CurrentEfficiency;
	monitoringvars.System.r_RountripEfficiency			:= monitor.system.r_RoundtripEfficiency;
	monitoringvars.System.s_SystemName					:= monitor.system.s_SystemName;
	monitoringvars.System.r_ChargedEnergy				:= monitor.powermonitor.BESS.r_EnergyConsumed;
	monitoringvars.System.r_DischargeEnergy				:= monitor.powermonitor.BESS.r_EnergySupplied;
	monitoringvars.System.b_Alert						:= GVL.b_WarningActive OR GVL.b_NormalShutdownActive OR GVL.b_QuickshutdownActive OR GVL.b_EmergencyShutdownActive OR NOT monitor.system.b_StartAllowed; 
	monitoringvars.System.b_TransportModePending		:= monitor.system.b_TransportModePending;

//AC DC charger
	monitoringvars.AcDcCharger.available				:= settings.Configuration.b_DcCharger AND monitor.AcDcCharger.by_NoModulesInstalled > 0;
	monitoringvars.AcDcCharger.r_AcPower				:= monitor.AcDcCharger.ACmeasurements.ar_ActivePower[0];
	monitoringvars.AcDcCharger.r_AcVoltage				:= monitor.AcDcCharger.ar_ACvoltage[0];
	monitoringvars.AcDcCharger.r_DcPower				:= monitor.AcDcCharger.r_DcPower;
	monitoringvars.AcDcCharger.state					:= TO_STRING(monitor.AcDcCharger.e_SystemStatus);	
	monitoringvars.AcDcCharger.r_AcCurrent				:= monitor.AcDcCharger.ACmeasurements.ar_Current[0];
	monitoringvars.AcDcCharger.r_AcCurrentMax			:= KwToCurrent(monitor.AcDcCharger.r_AvailablePower, monitor.AcDcCharger.ar_ACvoltage[0]);
	monitoringvars.AcDcCharger.r_AcPowerMax				:= monitor.AcDcCharger.r_AvailablePower;
			
//hystorize vars
	historizevars.Inverter.ActivePower					:=monitor.powerstack.r_Activepower;
	historizevars.Inverter.ReactivePower				:=monitor.powerstack.r_Reactivepower;
	historizevars.Inverter.Current						:=monitor.powerstack.r_ACcurrent;
	historizevars.Inverter.Voltage						:=monitor.powerstack.r_ACVoltageSupply;
	historizevars.Inverter.Frequency					:=monitor.powerstack.r_FrequencySupply;
	historizevars.Input.ActivePower						:=monitor.powermonitor.InputField.ar_ActivePower[0];
	historizevars.Input.ReactivePower					:=monitor.powermonitor.InputField.ar_ReactivePower[0];
	historizevars.Input.Current							:=monitor.powermonitor.InputField.ar_Current[0];
	historizevars.Input.Voltage							:=monitor.powermonitor.InputField.ar_LineVoltage[0];
	historizevars.Input.Frequency						:=monitor.powermonitor.InputField.ar_Frequency[0];
	historizevars.Output.ActivePower					:=monitor.powermonitor.OutputField.ar_ActivePower[0];
	historizevars.Output.ReactivePower					:=monitor.powermonitor.OutputField.ar_ReactivePower[0];
	historizevars.Output.Current						:=monitor.powermonitor.OutputField.ar_Current[0];
	historizevars.Output.Voltage						:=monitor.powermonitor.OutputField.ar_LineVoltage[0];
	historizevars.Output.Frequency						:=monitor.powermonitor.OutputField.ar_Frequency[0];
	historizevars.PSB.ActivePower						:=monitor.peakshavebox.Powermonitor.ar_ActivePower[0];
	historizevars.PSB.ReactivePower						:=monitor.peakshavebox.Powermonitor.ar_ReactivePower[0];
	historizevars.PSB.Current							:=monitor.peakshavebox.Powermonitor.ar_Current[0];
	historizevars.PSB.Voltage							:=monitor.peakshavebox.Powermonitor.ar_LineVoltage[0];
	historizevars.PSB.Frequency							:=monitor.peakshavebox.Powermonitor.ar_Frequency[0];
	historizevars.Battery.Current						:=monitor.battery.BatteryInfo.r_SystemCurrent;
	historizevars.Battery.Voltage						:=monitor.battery.BatteryInfo.r_SystemVoltage;
	historizevars.Battery.Power							:=monitor.battery.BatteryInfo.r_SystemPower;
	historizevars.Battery.SOC							:=monitor.battery.BatteryInfo.r_SocScaled;
	historizevars.Charger.ActivePower					:=monitor.AcDcCharger.ACmeasurements.ar_ActivePower[0];
	historizevars.Charger.ReactivePower					:=monitor.AcDcCharger.ACmeasurements.ar_ReactivePower[0];
	historizevars.Charger.Current						:=monitor.AcDcCharger.ACmeasurements.ar_Current[0];
	historizevars.Charger.Voltage						:=monitor.AcDcCharger.ar_ACvoltage[0];
	
//Powercontroller
	Monitoringvars.Powercontroller := monitor.system.PowerController;

//GengridController
	Monitoringvars.GenGridController := monitor.system.GenGridController;

//Switchgear
	Monitoringvars.Switchgear.b_NetContactorState 		:= monitor.powerstack.Netcontactor.b_NetConFb;
	Monitoringvars.Switchgear.b_ACInputState 			:= monitor.ACswitchgear.b_InputContactorfb AND monitor.ACswitchgear.b_InputMCCBfb;
	Monitoringvars.Switchgear.b_ACOutputState 			:= monitor.ACswitchgear.b_OutputMCCBfb;
	Monitoringvars.Switchgear.r_ACInputPower 			:= monitor.powermonitor.InputField.ar_Current[0];
	Monitoringvars.Switchgear.r_ACOutputPower 			:= monitor.powermonitor.OutputField.ar_Current[0];
	Monitoringvars.Switchgear.b_ACDetectedBusbar 		:= monitor.powerstack.b_ACDetected;
	Monitoringvars.Switchgear.b_ACDetectedInput 		:= monitor.powermonitor.InputField.e_ACrotationStatus <> 0;
	Monitoringvars.Switchgear.b_DCCouplingState 		:= monitor.DCswitchgear.b_CouplingState;
	Monitoringvars.Switchgear.b_DCDetected				:= monitor.battery.BatteryInfo.r_SystemVoltage > 120;
	Monitoringvars.Switchgear.r_DCCouplingCurrent 		:= monitor.DCswitchgear.r_Current;
	Monitoringvars.Switchgear.b_PeNeutralLink 			:= monitor.ACswitchgear.b_PENlinkfb;
	Monitoringvars.Switchgear.b_InputSync				:= monitor.ACswitchgear.b_InputSynchronizerfb;
	Monitoringvars.Switchgear.r_ACInputPower			:= monitor.powermonitor.InputField.ar_ActivePower[0];
	Monitoringvars.Switchgear.r_ACOutputPower			:= monitor.powermonitor.OutputField.ar_ActivePower[0];
	Monitoringvars.Switchgear.r_DCCouplingCurrent		:= 0; //monitor.powermonitor.DCbus.?

//Enclosure
	Monitoringvars.enclosure.b_DoorClosedClientPanel 	:= monitor.enclosure.doors.b_ClientpanelDoorClosed;
	Monitoringvars.enclosure.b_DoorClosedControlPanel	:= monitor.enclosure.doors.b_ControlPanelDoorClosed;
	Monitoringvars.enclosure.b_DoorClosedInverter		:= monitor.safety.b_InverterDoorOK;
	Monitoringvars.enclosure.b_HumidityHigh				:= monitor.enclosure.climate.events.b_HumidityHigh;
	Monitoringvars.enclosure.b_HumidityTooHigh			:= monitor.enclosure.climate.events.b_HumidityTooHigh;
	Monitoringvars.enclosure.b_TemperatureHigh			:= monitor.enclosure.climate.events.b_TemperatureHigh;
	Monitoringvars.enclosure.b_TemperatureTooHigh 		:= monitor.enclosure.climate.events.b_TemperatureTooHigh;
	Monitoringvars.enclosure.b_TemperatureLow 			:= monitor.enclosure.climate.events.b_TemperatureLow;
	Monitoringvars.enclosure.b_TemperatureTooLow 		:= monitor.enclosure.climate.events.b_TemperatureTooLow;
	Monitoringvars.enclosure.r_Humidity					:= monitor.enclosure.climate.r_Humidity;
	Monitoringvars.enclosure.r_Temperature 				:= monitor.enclosure.climate.r_Temperature;
	
//Firedetection
	Monitoringvars.firedetection.e_SmokeDetectorState 	:= monitor.protections.FireDetection.SmokeDetectors.State;
	Monitoringvars.firedetection.e_CoDetectorState 		:= monitor.protections.FireDetection.CoDetectors.State;
	Monitoringvars.firedetection.r_CoDetectorLeftValue 	:= monitor.protections.FireDetection.CoDetectors.Value[1];
	Monitoringvars.firedetection.r_CoDetectorRightValue := monitor.protections.FireDetection.CoDetectors.Value[2];
	
//Overcurrent protection
	monitoringvars.OCP.b_InputMCCBstate					:= monitor.ACswitchgear.b_InputMCCBfb;
	monitoringvars.OCP.b_OutputMCCBstate				:= monitor.ACswitchgear.b_OutputMCCBfb;
	monitoringvars.OCP.b_InputOverloadAlarm 			:= monitor.protections.OvercurrentProtection.b_InputAlarm;
	monitoringvars.OCP.b_OutputOverloadAlarm 			:= monitor.protections.OvercurrentProtection.b_OutputAlarm;
	monitoringvars.OCP.b_InputOverloadWarning 			:= monitor.protections.OvercurrentProtection.b_InputWarning;
	monitoringvars.OCP.b_OutputOverloadWarning 			:= monitor.protections.OvercurrentProtection.b_OutputWarning;
	monitoringvars.OCP.r_CurrentPeak 					:= monitor.protections.OvercurrentProtection.r_PeakCurrent;
	monitoringvars.OCP.s_Location 						:= monitor.protections.OvercurrentProtection.s_locationPeak;
	monitoringvars.OCP.t_PeakDuration 					:= monitor.protections.OvercurrentProtection.t_PeakCurrentDuration;
	
//protections
	monitoringvars.protections.b_InsulationOk 			:= monitor.safety.b_InsulationMonitorOK;
	monitoringvars.protections.e_EarthingSystemDetected := monitor.protections.Insulation.e_EarthingSystemDetected;
	monitoringvars.protections.b_InsulationAlarm 		:= NOT monitor.safety.b_InsulationMonitorOK;
	monitoringvars.protections.b_InsulationPenDetected 	:= monitor.protections.Insulation.b_PENlinkDetected;
	monitoringvars.protections.b_InsulationEnable 		:= monitor.protections.Insulation.b_Enabled;
	monitoringvars.protections.b_InsulationWarning 		:= monitor.protections.Insulation.b_Warning;
	monitoringvars.protections.b_MrcdbWarning			:= monitor.protections.MRCDB.b_prewarning;
	monitoringvars.protections.b_MrcdbOK 				:= monitor.safety.b_MRCDBOK;
	monitoringvars.protections.b_MrcdbAlarm 			:= NOT monitor.safety.b_MRCDBOK;
	monitoringvars.protections.b_SurgeType12OK 			:= monitor.protections.Surge.b_Type12_OK;
	monitoringvars.protections.b_SurgeType3OK 			:= monitor.protections.Surge.b_Type3_OK;

	
//UPS
	monitoringvars.UPS.b_BatteryLowCritical				:= monitor.internalpsu.UPS.Events.b_BatteryLowError;
	monitoringvars.UPS.b_BatteryLowWarning				:= monitor.internalpsu.UPS.Events.b_BatteryLowWarning;
	monitoringvars.UPS.b_BatteryLowInfo					:= monitor.internalpsu.UPS.Events.b_BatteryLowInfo;
	monitoringvars.UPS.b_ChargerActive					:= monitor.internalpsu.UPS.b_ChargerActive;
	monitoringvars.UPS.b_InputVoltageFault				:= monitor.internalpsu.UPS.Events.b_InputVoltageWarning;
	monitoringvars.UPS.b_SupplyOnBattery				:= monitor.internalpsu.UPS.b_SystemOnBattery;
	monitoringvars.UPS.r_BatteryVoltage					:= monitor.internalpsu.UPS.r_BatteryVoltage;
	monitoringvars.UPS.r_InputVoltage					:= monitor.internalpsu.UPS.r_InputVoltage;
	monitoringvars.UPS.r_OutputVoltage					:= monitor.internalpsu.UPS.r_OutputVoltage;
	monitoringvars.UPS.r_OutputCurrent					:= monitor.internalpsu.UPS.r_OutputCurrent;
	monitoringvars.UPS.ui_SoC							:= monitor.internalpsu.UPS.ui_SOC;
	
//Internal powersupply
	monitoringvars.IPSU.b_24VdcOK						:= monitor.internalpsu.b_24VdcAvailable;
	monitoringvars.IPSU.b_400VacOK						:= monitor.internalpsu.b_400VACAvailable;
	monitoringvars.IPSU.b_HvdcOK						:= monitor.internalpsu.b_HVDCAvailable;
	monitoringvars.IPSU.e_400VSource					:= monitor.internalpsu.e_400VSupplySource;
	monitoringvars.IPSU.b_CeeFuseOK						:= NOT(monitor.internalpsu.Events.b_CEEInputFuseTripped);
	monitoringvars.IPSU.b_GridFuseOK					:= NOT(monitor.internalpsu.Events.b_GridInputFuseTripped);
	
//Zeropoint transformer
	monitoringvars.ZPT.b_ZPTOverloadAlarm				:= monitor.neutraltransformer.events.b_OvercurrentAlarm OR monitor.neutraltransformer.events.b_NeutralCurrentTooHigh;
	monitoringvars.ZPT.b_ZPTOverloadWarning				:= monitor.neutraltransformer.events.b_OvercurrentWarning OR monitor.neutraltransformer.events.b_NeutralCurrentHigh;
	monitoringvars.ZPT.b_VoltageUnbalanceAlarm			:= monitor.neutraltransformer.events.b_VoltageUnbalanceTooHigh;
	monitoringvars.ZPT.b_VoltageUnbalanceWarning		:= monitor.neutraltransformer.events.b_VoltageUnbalanceHigh;
	monitoringvars.ZPT.r_TemperatureL1					:= monitor.neutraltransformer.r_TemperaturePhase[1];
	monitoringvars.ZPT.r_TemperatureL2					:= monitor.neutraltransformer.r_TemperaturePhase[2];
	monitoringvars.ZPT.r_TemperatureL3					:= monitor.neutraltransformer.r_TemperaturePhase[3];
	monitoringvars.ZPT.r_voltageunbalance				:= monitor.powermonitor.OutputField.r_VoltageUnbalance;
	monitoringvars.ZPT.r_powerload						:= monitor.neutraltransformer.r_Powerload;
	monitoringvars.ZPT.b_TempWarningL1					:= monitor.neutraltransformer.events.b_TemperatureHighPhase[1];
	monitoringvars.ZPT.b_TempWarningL2					:= monitor.neutraltransformer.events.b_TemperatureHighPhase[2];
	monitoringvars.ZPT.b_TempWarningL3					:= monitor.neutraltransformer.events.b_TemperatureHighPhase[3];
	monitoringvars.ZPT.b_TempAlarmL1					:= monitor.neutraltransformer.events.b_TemperatureTooHighPhase[1];
	monitoringvars.ZPT.b_TempAlarmL2					:= monitor.neutraltransformer.events.b_TemperatureTooHighPhase[2];
	monitoringvars.ZPT.b_TempAlarmL3					:= monitor.neutraltransformer.events.b_TemperatureTooHighPhase[3];

//connections
	monitoringvars.Connections.b_IoTEnabled				:= Iotcontrolvars.b_Active;
	monitoringvars.Connections.e_IoTConnectionState		:= IoTcontrolvars.e_ConnectionState;
	monitoringvars.Connections.b_ExtControllerEnabled	:= PNcontrolvars.b_Active;
	monitoringvars.Connections.e_ExtConnectionState		:= PNcontrolvars.e_ConnectionState;
	monitoringvars.Connections.s_OutputJson				:= PNcontrolvars.s_OutputJson;
	monitoringvars.Connections.b_PsbOK					:= monitor.peakshavebox.b_buscouplerReady;
	monitoringvars.Connections.e_ActiveController		:= controlvars.HardSettings.setup.e_ControlSource;
	monitoringvars.Connections.e_EthercatState			:= monitor.PLC.e_EthercatState;
	monitoringvars.Connections.e_ProfinetState			:= monitor.PLC.e_ProfinetState;
	monitoringvars.Connections.r_CPUload				:= monitor.PLC.r_CPUload;
	
//battery
	monitoringvars.Battery.r_SoCReal					:= monitor.battery.BatteryInfo.r_SOC;
	monitoringvars.Battery.e_status						:= monitor.battery.BatteryInfo.e_BMS_Status;
	monitoringvars.Battery.r_SocScaled					:= monitor.battery.BatteryInfo.r_SOCScaled;
	monitoringvars.Battery.r_MaxDischargePower			:= monitor.battery.BatteryInfo.r_MaxDischargePowerAllowed;
	monitoringvars.Battery.r_MaxChargePower				:= monitor.battery.BatteryInfo.r_MaxChargePowerAllowed;
	monitoringvars.Battery.r_CellTempMin				:= monitor.battery.BatteryInfo.ar_CellTemperature[eSubValues.Minimum];
	monitoringvars.Battery.r_CellTempMax				:= monitor.battery.BatteryInfo.ar_CellTemperature[eSubValues.Maximum];													
	monitoringvars.Battery.r_CellVoltageMin				:= monitor.battery.BatteryInfo.ar_CellVoltage[eSubValues.Minimum];
	monitoringvars.Battery.r_CellVoltageMax				:= monitor.battery.BatteryInfo.ar_CellVoltage[eSubValues.Maximum];								
	monitoringvars.Battery.r_SoH						:= monitor.battery.BatteryInfo.r_SOH;
	monitoringvars.Battery.r_DCcurrent					:= monitor.battery.BatteryInfo.r_SystemCurrent;
	monitoringvars.Battery.r_DCvoltage					:= monitor.battery.BatteryInfo.r_SystemVoltage;
	monitoringvars.Battery.r_NetRemainingCapacity		:= monitor.battery.BatteryInfo.r_RemainingDischargeEnergyNett;
	monitoringvars.Battery.ui_CycleCount				:= monitor.battery.BatteryInfo.ui_CycleCount;
	
//Powerstack
	monitoringvars.Powerstack.b_ACDetected				:= monitor.powerstack.b_GridACdetected;
	monitoringvars.Powerstack.b_DCDetected				:= monitor.powerstack.b_DCDetected;
	monitoringvars.Powerstack.b_StartedState			:= monitor.powerstack.b_StartedState;
	monitoringvars.Powerstack.b_ControlEnabled			:= monitor.powerstack.b_ControlEnabled;
	monitoringvars.Powerstack.b_MasterEnabled			:= monitor.powerstack.PowermoduleMaster.b_online;
	monitoringvars.Powerstack.b_SlaveEnabled			:= monitor.powerstack.PowermoduleSlave.b_online AND settings.Configuration.b_DoublePowerModule;
	monitoringvars.Powerstack.r_ActivePower				:= monitor.powerstack.r_ActivePower;
	monitoringvars.Powerstack.r_DcPower					:= monitor.powerstack.r_Dcpower;
	monitoringvars.Powerstack.r_Powerload				:= monitor.powerstack.r_LoadPercent;
	monitoringvars.Powerstack.e_MasterState				:= monitor.powerstack.Powermodulemaster.e_Status;
	monitoringvars.Powerstack.e_SlaveState				:= monitor.powerstack.Powermoduleslave.e_Status;
	monitoringvars.Powerstack.b_MasterCurrThrotActive	:= monitor.powerstack.PowermoduleMaster.Events.b_CurrThrottlingActive;
	monitoringvars.Powerstack.b_MasterTempThrotActive	:= monitor.powerstack.PowermoduleMaster.Events.b_TempThrottlingActive;
	monitoringvars.Powerstack.r_MasterthrotValue		:= monitor.powerstack.PowermoduleMaster.r_OverCurrentValue;
	monitoringvars.Powerstack.b_MasterWarning			:= monitor.powerstack.Events.b_MasterWarning;
	monitoringvars.Powerstack.b_MasterMCCBfb			:= monitor.powerstack.PowermoduleMaster.b_MccbFb;
	monitoringvars.Powerstack.b_SlaveCurrThrotActive	:= monitor.powerstack.PowermoduleSlave.Events.b_CurrThrottlingActive;
	monitoringvars.Powerstack.b_SlaveTempThrotActive	:= monitor.powerstack.PowermoduleSlave.Events.b_TempThrottlingActive;
	monitoringvars.Powerstack.r_SlavethrotValue			:= monitor.powerstack.PowermoduleSlave.r_OverCurrentValue;
	monitoringvars.Powerstack.b_SlaveWarning			:= monitor.powerstack.Events.b_SlaveWarning;
	monitoringvars.Powerstack.b_SlaveMCCBfb				:= monitor.powerstack.PowermoduleSlave.b_MccbFb;
	monitoringvars.Powerstack.r_throttlingValue			:= monitor.powerstack.r_OvercurrentValueAct;
	monitoringvars.Powerstack.e_NetContState			:= monitor.powerstack.Netcontactor.e_NetConState;
	monitoringvars.powerstack.e_StatusPowerStack		:= monitor.powerstack.e_State;
	monitoringvars.Powerstack.e_ACrotationState			:= monitor.powermonitor.OutputField.e_ACrotationStatus;
	monitoringvars.Powerstack.b_islandOperation			:= monitor.powerstack.b_InverterGridFormingMode;
	
//Coolingsystem
	monitoringvars.cooling.e_OperationMode 				:= monitor.Cooling.CoolingSystemMode;
	monitoringvars.cooling.r_CoolantPressure			:= monitor.Cooling.r_CoolantPressure;
	monitoringvars.cooling.r_CoolantTemperature			:= monitor.Cooling.r_CoolantTemperature;
	monitoringvars.cooling.r_EnclosureDewpoint			:= monitor.Cooling.r_EnclosureDewpoint;
	monitoringvars.cooling.e_HeatPumpStatus				:= monitor.Cooling.HeatPumpStatus;
	monitoringvars.cooling.b_HeatPumpError				:= monitor.Cooling.Events.b_HeatpumpWarning;
	monitoringvars.cooling.b_HeatPumpWarning			:= monitor.Cooling.Events.b_HeatpumpError;
	monitoringvars.cooling.b_CoolantPressureError		:= monitor.Cooling.Events.b_CoolingLoopIdlePressureError OR monitor.Cooling.Events.b_InverterCoolingLoopError;
	monitoringvars.cooling.b_CoolantPressureWarning		:= monitor.Cooling.Events.b_CoolingLoopIdlePressureWarning;
	monitoringvars.cooling.b_CoolantTempWarning			:= monitor.Cooling.Events.b_SystemOvertemperatureWarning OR monitor.Cooling.Events.b_SystemUndertemperatureWarning;
	
//control feedback
	monitoringvars.controlfb 							:= monitor.controlfb.control;
	
//limits
	monitoringvars.Limits.r_ACcurrentLimit				:= 650;
	monitoringvars.Limits.r_ApparentPowerlimit			:= 450;
	monitoringvars.Limits.r_ActivePowerlimit			:= 360;
	monitoringvars.Limits.r_DCcurrentLimit				:= monitor.battery.BatteryInfo.r_ratedCurrent;
	monitoringvars.limits.r_DroopLimit 					:= settings.MachineParams.Powerstack.r_DroopMaximum;
	
//ConditionalFormatting
	ConditionalFormatting(monitoringvars.ConditionalFormatting, controlvars);
	
//PSB
	monitoringvars.PSB.b_Connected 						:= monitor.peakshavebox.b_buscouplerReady;
	monitoringvars.PSB.b_Active							:= monitor.peakshavebox.b_active;
END_ACTION

METHOD ResetControlvarsOnVariant : BOOL
VAR_INPUT
END_VAR
IF NOT settings.Configuration.b_ACInputConnection THEN
	controlvars.SoftSettings.setup.e_AcInputType := eACInputType.None;
END_IF
END_METHOD

METHOD ResetHMIvarsOnEvent

VAR_INST
	
END_VAR
rTrigResetPowerSetpoints(CLK:= NOT monitor.powerstack.b_StartedState); //monitor.controlfb.HardSettings.setup.e_ControlSource <> 0 OR monitor.system.e_gridmode <> eGridmode.forming);

IF rTrigResetPowerSetpoints.Q THEN
	Controlvars.Operation.system.r_PFset := 1;
	controlvars.Operation.system.r_Pset := 0;
	controlvars.Operation.system.r_Qset := 0;
	controlvars.control.b_start := FALSE;
	controlvars.control.b_stop := FALSE;
END_IF

IF monitor.controlfb.Operation.system.b_GridTakeOverEnable AND monitor.powerstack.b_InverterGridFormingMode THEN
	controlvars.Operation.system.r_Pset := monitor.powerstack.r_ActivePower;
END_IF
END_METHOD

METHOD SetArraydata : BOOL

VAR_IN_OUT
	arrays			: ST_HMI_Monitor_Arraydata;
	init			: BOOL;
END_VAR

VAR_INPUT
	b_sync			: BOOL;
END_VAR

VAR
	index				: INT ;	
END_VAR
IF b_sync OR init THEN
	FOR index := 1 TO (SIZEOF(Arrays.ACInputData) / SIZEOF(st_HMIData)) DO
		DataToHMIArrayFormat(data:= GetAcInputArrayData(data := monitor.powermonitor.inputfield, id:=index), init:= init, st_DataOut := arrays.ACInputData[index]);
	END_FOR
	FOR index := 1 TO (SIZEOF(Arrays.ACOutputData) / SIZEOF(st_HMIData)) DO
		DataToHMIArrayFormat(data:= GetAcOutputArrayData(data := monitor.powermonitor.OutputField, id:=index), init:= init, st_DataOut := arrays.ACOutputData[index]);
	END_FOR
	FOR index := 1 TO (SIZEOF(Arrays.PowerstackData) / SIZEOF(st_HMIData)) DO
		DataToHMIArrayFormat(data:= GetPowerstackArrayData(id:=index), init:= init, st_DataOut := arrays.PowerstackData[index]);
	END_FOR
	FOR index := 1 TO (SIZEOF(Arrays.PmMasterData) / SIZEOF(st_HMIData)) DO
		DataToHMIArrayFormat(data:= GetPowerModuleArrayData(data := monitor.powerstack.PowermoduleMaster, id:=index), init:= init, st_DataOut := arrays.PmMasterData[index]);
	END_FOR
	IF settings.Configuration.b_DcCharger OR INIT THEN
		FOR index := 1 TO (SIZEOF(Arrays.AcDcChargerData) / SIZEOF(st_HMIData)) DO
			DataToHMIArrayFormat(data:= GetDcChargerData(data := monitor.AcDcCharger, id:=index), init:= init, st_DataOut := arrays.AcDcChargerData[index]);
		END_FOR
	END_IF
	IF settings.Configuration.b_DCbuscoupling OR INIT THEN
		FOR index := 1 TO (SIZEOF(Arrays.DcExtension) / SIZEOF(st_HMIData)) DO
			DataToHMIArrayFormat(data:= GetDcExtData(data := monitor.DCswitchgear, id:=index), init:= init, st_DataOut := arrays.DcExtension[index]);
		END_FOR
	END_IF
	IF settings.Configuration.b_DoublePowerModule THEN
		FOR index := 1 TO (SIZEOF(Arrays.PmSlaveData) / SIZEOF(st_HMIData)) DO
			DataToHMIArrayFormat(data:= GetPowerModuleArrayData(data := monitor.powerstack.PowermoduleSlave, id:=index), init:= init, st_DataOut := arrays.PmSlaveData[index]);
		END_FOR
	END_IF
	IF settings.MachineParams.GenComm.GenControlProtocol <> 0 OR init THEN
		FOR index := 1 TO (SIZEOF(Arrays.Genset) / SIZEOF(st_HMIData)) DO
			DataToHMIArrayFormat(data:= GetGensetData(data := monitor.Generator, id:=index), init:= init, st_DataOut := arrays.Genset[index]);
		END_FOR
	END_IF
	FOR index := 1 TO (SIZEOF(Arrays.PNcontrolData) / SIZEOF(st_HMIData)) DO
		DataToHMIArrayFormat(data:= GetextcontrolData(data := Pncontrolvars, id:=index), init:= init, st_DataOut := arrays.PNcontrolData[index]);
	END_FOR
	
	FOR index := 1 TO (SIZEOF(Arrays.iotcontrolData) / SIZEOF(st_HMIData)) DO
		DataToHMIArrayFormat(data:= GetextcontrolData(data := IOtcontrolvars, id:=index), init:= init, st_DataOut := arrays.IotcontrolData[index]);
	END_FOR
	FOR index := 1 TO (SIZEOF(Arrays.PSBData) / SIZEOF(st_HMIData)) DO
		DataToHMIArrayFormat(data:= GetPSBData(data := Monitor.peakshavebox, id:=index), init:= init, st_DataOut := arrays.PSBData[index]);
	END_FOR
	FOR index := 1 TO (SIZEOF(Arrays.MBMUdata) / SIZEOF(st_HMIData)) DO
		DataToHMIArrayFormat(data:= GetMBMUData(data := monitor.battery.BatteryInfo, id:=index), init:= init, st_DataOut := arrays.MBMUdata[index]);
	END_FOR
	FOR index := 1 TO (SIZEOF(Arrays.SBMU1data) / SIZEOF(st_HMIData)) DO
		DataToHMIArrayFormat(data:= GetSBMUData(data := monitor.battery.SBMU[0], id:=index, 1), init:= init, st_DataOut := arrays.SBMU1data[index]);
	END_FOR
	FOR index := 1 TO (SIZEOF(Arrays.SBMU2data) / SIZEOF(st_HMIData)) DO
		DataToHMIArrayFormat(data:= GetSBMUData(data := monitor.battery.SBMU[1], id:=index, 2), init:= init, st_DataOut := arrays.SBMU2data[index]);
	END_FOR
	FOR index := 1 TO (SIZEOF(Arrays.SBMU3data) / SIZEOF(st_HMIData)) DO
		DataToHMIArrayFormat(data:= GetSBMUData(data := monitor.battery.SBMU[2], id:=index, 3), init:= init, st_DataOut := arrays.SBMU3data[index]);
	END_FOR
	FOR index := 1 TO (SIZEOF(Arrays.SBMU4data) / SIZEOF(st_HMIData)) DO
		DataToHMIArrayFormat(data:= GetSBMUData(data := monitor.battery.SBMU[3], id:=index, 4), init:= init, st_DataOut := arrays.SBMU4data[index]);
	END_FOR
	FOR index := 1 TO (SIZEOF(Arrays.CoolingSystem) / SIZEOF(st_HMIData)) DO
		DataToHMIArrayFormat(data:= GetCoolingData(data := monitor.Cooling, id:=index), init:= init, st_DataOut := arrays.CoolingSystem[index]);
	END_FOR
	FOR index := 1 TO (SIZEOF(Arrays.CoolingSystemHp1) / SIZEOF(st_HMIData)) DO
		DataToHMIArrayFormat(data:= GetHeatpumpData(data := monitor.Cooling.HeatPumpSystem.PrimaryHeatpumpGet, id:=index), init:= init, st_DataOut := Arrays.CoolingSystemHp1[index]);
	END_FOR
	FOR index := 1 TO (SIZEOF(Arrays.CoolingSystemHp2) / SIZEOF(st_HMIData)) DO
		DataToHMIArrayFormat(data:= GetHeatpumpData(data := monitor.Cooling.HeatPumpSystem.SecondaryHeatpumpGet, id:=index), init:= init, st_DataOut := Arrays.CoolingSystemHp2[index]);
	END_FOR
	
END_IF
END_METHOD

METHOD SettingsChanged : BOOL

VAR_INPUT
	adr1		: DWORD;
	adr2		: DWORD;
	size		: DWORD;
END_VAR

//VAR_IN_OUT CONSTANT
//	hs_user					: ST_hardsettings;
//	hs_PLC					: ST_hardsettings;
	
//END_VAR
SettingsChanged := (MEMCMP(adr1, adr2, size) <> 0);
END_METHOD

END_PROGRAM

// ---- POUs/MonitoringControl/HMI/FB_HMIButtons.TcPOU
FUNCTION_BLOCK FB_HMIButtons
VAR_IN_OUT
	controlvars				: ST_HMI_control;
	monitoringvars			: ST_HMI_monitor;
END_VAR
VAR_INPUT
	b_ControlAccess			: BOOL;
END_VAR
VAR
	DemoModeTimer				: TON := (PT := T#3s);
	b_StopButton		AT %I* : BOOL;
	b_StopButtonLight	AT %Q* : BOOL;
	b_Button			AT %I* : ARRAY [1..6] OF BOOL;
	b_ButtonLight		AT %Q* : ARRAY [1..6] OF BOOL;
	
	fbQsetbyStep					: FB_IncrementPowerStep;
	fbPsetbyStep					: FB_IncrementPowerStep;
	
	b_FlashSlow						: BOOL;
	b_FlashQuick					: BOOL;
END_VAR

PulseLampTriggers();

fbPsetbyStep(
	b_Up := controlvars.HMIonly.b_Pup,
	b_Down:= controlvars.HMIonly.b_Pdown,
	b_Reset:= controlvars.HMIonly.b_PReset,
	r_IncrementStep := 5,
	r_power	:= controlvars.Operation.system.r_Pset);
		
fbQsetbyStep(
	b_Up := controlvars.HMIonly.b_Qup,
	b_Down:= controlvars.HMIonly.b_Qdown,
	b_Reset:= controlvars.HMIonly.b_QReset,
	r_IncrementStep := 5,
	r_power	:= controlvars.Operation.system.r_Qset);
	
controlvars.control.b_SystemShutdown := StopButton(b_in := b_stopButton AND b_ControlAccess, b_lamp=>b_stopButtonLight);

//LED DEMO TRIGGER
DemoModeTimer(IN :=  b_Button[4] AND b_Button[3] AND NOT DemoModeTimer.Q);
IF DemoModeTimer.Q THEN
	GVL.b_LEDDemoMode := NOT GVL.b_LEDDemoMode;
END_IF

//Reset
ResetButton(IN := b_Button[5], variable := controlvars.control.b_Reset, b_lamp =>b_ButtonLight[5]);

//Mute Sounder
SounderMuteButton(IN := b_Button[6] AND b_ControlAccess, variable := controlvars.Operation.system.b_SounderMute);

//Transportmode
TransportMode(IN := b_Button[1], b_lamp => b_ButtonLight[1], b_TransportmodeEnable := controlvars.SoftSettings.system.b_EnableTransportMode);
Monitoringvars.ConditionalFormatting.b_TransportModeActive := b_ButtonLight[1];

METHOD HMIStartEnd : BOOL
VAR_INPUT
	b_taskKill	: BOOL;
END_VAR

VAR_INST
	fbHMIstart : NT_StartProcess;
	b_hmistart	: BOOL := FALSE;
	ton_HmiStart: TON;
	fbTaskKill	: NT_StartProcess;
END_VAR
//HMI autostart on PLC. Only needed when nuc is not installed.
ton_HMIstart(IN:= b_hmiStart, PT:= T#20S);
fbHMIstart(
	NETID		:= '',
	PATHSTR		:= 'C:\Program Files\Google\Chrome\Application\chrome.exe',
	DIRNAME		:= 'C:\Program Files\Google\Chrome\Application',
	COMNDLINE	:= '--chrome-frame  --kiosk https://127.0.0.1:1020',
	START		:= ton_HMIstart.Q,
	TMOUT		:= T#5S,
);

IF fbHMIstart.BUSY THEN
	b_hmistart := FALSE;
END_IF

//Exit kiosk mode
fbTaskKill(
	NETID		:= '',
	PATHSTR		:= 'C:\PLCUtility\CloseHMI.bat',
	DIRNAME		:= 'C:\PLCUtility',
	COMNDLINE	:= '',
	START		:= b_taskKill,
	TMOUT		:= T#5S,
);

IF fbTaskKill.BUSY THEN
	b_taskKill := FALSE;
END_IF
END_METHOD

METHOD PulseLampTriggers : BOOL
VAR_INPUT
END_VAR
VAR_INST
	ton_FlashPulseQuick					: TON := (PT := T#250MS);
	ton_FlashPulseSlow					: TON := (PT := T#500MS);
END_VAR
ton_flashPulseQuick(IN:= NOT ton_flashPulseQuick.Q );
IF ton_FlashPulseQuick.Q THEN
	b_FlashQuick := NOT b_FlashQuick;
END_IF

ton_flashPulseSlow(IN:= NOT ton_flashPulseSlow.Q );
IF ton_FlashPulseSlow.Q THEN
	b_FlashSlow := NOT b_FlashSlow;
END_IF
END_METHOD

METHOD ResetButton
VAR_INPUT
	IN				: BOOL;
END_VAR

VAR_IN_OUT
	variable			: BOOL;
END_VAR

VAR_INST
	f_Trig		: F_TRIG;
END_VAR

VAR_OUTPUT
	b_lamp			: BOOL;
END_VAR
f_Trig(CLK := IN);

IF IN THEN
	variable := IN;
END_IF

IF f_Trig.Q THEN
	variable := FALSE;
END_IF

b_lamp := GVL.b_EmergencyShutdownActive OR GVL.b_NormalShutdownActive;
END_METHOD

METHOD SounderMuteButton
VAR_INPUT
	IN				: BOOL;
END_VAR

VAR_IN_OUT
	variable			: BOOL;
END_VAR

VAR_INST
	f_Trig			: F_TRIG;
END_VAR
f_Trig(CLK := IN);

IF IN THEN
	variable := IN;
END_IF

IF f_Trig.Q THEN
	variable := FALSE;
END_IF
END_METHOD

METHOD StopButton : BOOL
VAR_INPUT
	b_in : BOOL;
END_VAR

VAR_OUTPUT
	b_lamp : BOOL;
END_VAR

VAR_INST
	ton_ShutdownDelay	: TON := (PT := T#3S);
END_VAR
//Set systemshutdown
ton_ShutdownDelay(IN := b_IN);
StopButton := ton_ShutdownDelay.Q;


//Set lamp based on mode.
IF monitoringvars.system.e_SystemState = eSystemstate.Shutdown THEN
	b_lamp := b_FlashQuick;
ELSIF monitoringvars.system.e_SystemState <> eSystemstate.off THEN
	b_lamp := b_FlashSlow AND b_IN;
END_IF
END_METHOD

METHOD TransportMode
VAR_INPUT
	IN				: BOOL;
END_VAR

VAR_OUTPUT
	b_lamp			: BOOL;
END_VAR

VAR_IN_OUT
	b_TransportmodeEnable	: Bool;
END_VAR

VAR_INST
	r_trigbutton : r_TRIG;
END_VAR
r_trigbutton(CLK:= IN);

IF r_trigbutton.Q THEN
	b_transportmodeEnable := NOT b_transportmodeEnable;
END_IF

IF monitoringvars.System.b_TransportModePending THEN
	b_lamp := b_FlashSlow;
ELSE
	b_lamp := b_transportmodeEnable;
END_IF
END_METHOD

END_FUNCTION_BLOCK

// ---- POUs/Functions-FBs-Programs/fb_IncrementPowerStep.TcPOU
FUNCTION_BLOCK fb_IncrementPowerStep
VAR_INPUT
	b_Up			: BOOL;
	b_Down			: BOOL;
	b_Reset			: BOOL;
	r_incrementStep	: REAL:= 5;
END_VAR

VAR_IN_OUT
	r_Power			: REAL;
END_VAR

VAR
	ton_IncrementPulse				: TON := (PT := T#1S);
	tof_MaxContinuesIncrementTime 	: TOF := (PT := T#10S);
	r_TrigUpDown					: r_Trig;
END_VAR

tof_MaxContinuesIncrementTime(IN:= b_Up OR b_Down);
ton_incrementPulse(IN := NOT(ton_incrementpulse.Q) AND (b_Up OR b_Down));
r_trigUpDown(CLK:= b_Up OR b_Down);

IF (r_trigUpDown.Q OR ton_incrementPulse.Q) AND tof_MaxContinuesIncrementTime.Q THEN
	IF (b_UP AND NOT b_Down) THEN
		r_Power := r_Power + r_IncrementStep;
	ELSIF (NOT b_UP AND b_Down) THEN
		r_Power := r_Power - r_IncrementStep;
	END_IF
END_IF

IF b_reset THEN
	r_Power := 0;
END_IF

END_FUNCTION_BLOCK

// ---- POUs/Functions-FBs-Programs/_acFunctions/kWToCurrent.TcPOU
FUNCTION kWToCurrent : REAL
VAR_INPUT
	kw			: REAL;
	linevoltage	: REAL;
END_VAR

IF linevoltage > 100 THEN
	kWToCurrent := kw *1000 / (linevoltage * 1.73);
ELSE
	kWToCurrent := kw *1000 / (400 * 1.73);
END_IF

END_FUNCTION

// ---- POUs/Functions-FBs-Programs/_acFunctions/ReactivePower.TcPOU
FUNCTION ReactivePower : Real
VAR_INPUT
	AppPower	: REAL;
	RealPower 	: REAL;
	PowerFactor	: REAL;
END_VAR
VAR
END_VAR

IF RealPower > AppPower THEN // NAN solution
	RETURN;
END_IF

IF powerfactor < 0 THEN
	ReactivePower := - SQRT(EXPT(AppPower, 2) - EXPT(RealPower,2));
ELSE
	ReactivePower := SQRT(EXPT(AppPower, 2) - EXPT(RealPower,2));
END_IF

END_FUNCTION

// ---- POUs/Functions-FBs-Programs/_acFunctions/PowerFactor.TcPOU
FUNCTION PowerFactor : REAL
VAR_INPUT
	r_P	: REAL;
	r_S	: REAL;
	r_Q	: REAL;
END_VAR

VAR
	PFRaw	: REAL;
	Factor	: INT;
END_VAR

PFRaw := ABS(r_P) / MAX(0.001, ABS(r_S));
Factor := SEL(r_Q < 0, -1, 1);

Powerfactor := LIMIT(-1, PFRaw * Factor, 1);

END_FUNCTION

// ---- POUs/System/FB_SystemControl.TcPOU
FUNCTION_BLOCK FB_SystemControl
VAR_IN_OUT
	st_params								: ST_System_params;
	st_calibration							: ST_System_calibration;
	monitor								   	: ST_System_Monitor;
	control									: ST_System_Control;
END_VAR

VAR
	//fbs
	b_calibrationRunning					: BOOL;
	PowerControl							: FB_PowerControl;
	GenGridControl							: FB_GenGridController;
	r_trigStoreMachineSettings				: R_TRIG;
	
	b_skipPowerTest								: BOOL := TRUE;
	b_StoreMachineSettings						: BOOL;
	b_loadonly									: BOOL;
	sMessage									: STRING;	

	buffer										: ARRAY [0..24] OF WORD;		

END_VAR

VAR_OUTPUT
	toSystem								: ST_System_set();
END_VAR

//call methods
CalculateEfficiency(
	powerstack := monitor.powerstack, 
	powermonitor := monitor.powermonitor, 
	system := monitor.system,
	battery := monitor.battery);
	
FillSystemMonitoringVars();

MapUsercontrolsToSystemVars();

GetEvents();

//store machine settings
r_trigStoreMachineSettings(CLK := settings.Save OR settings.Load);
IF r_trigStoreMachineSettings.Q THEN
	b_StoreMachineSettings := TRUE;
END_IF

IF b_StoreMachineSettings AND_THEN storeSettings(TRUE, settings.Save) THEN;
	b_StoreMachineSettings := FALSE;
END_IF

//calibration script
IF NOT st_calibration.Powerstack.Slave.b_StartCalibration THEN
	PowerstackCalibration(start := st_calibration.Powerstack.Master.b_StartCalibration, skippowertest := b_skipPowerTest, loadonly := b_loadonly,   
		powerstack := monitor.powerstack,
		powermoduleCalib := st_calibration.Powerstack.Master,
		PMeasured := monitor.powermonitor.OutputField.ar_ActivePower[0],
		QMeasured := monitor.powermonitor.OutputField.ar_ReactivePower[0],
		sMessage => sMessage);
ELSIF NOT st_calibration.Powerstack.Master.b_StartCalibration THEN
	PowerstackCalibration(start := st_calibration.Powerstack.Slave.b_StartCalibration, skippowertest := b_skipPowerTest, loadonly := b_loadonly,   
		powerstack := monitor.powerstack,
		powermoduleCalib := st_calibration.Powerstack.Slave,
		PMeasured := monitor.powermonitor.OutputField.ar_ActivePower[0],
		QMeasured := monitor.powermonitor.OutputField.ar_ReactivePower[0],
		sMessage => sMessage);
END_IF
b_calibrationRunning := settings.Calibration.Powerstack.Master.b_StartCalibration OR settings.Calibration.Powerstack.Slave.b_StartCalibration;


UpdateSystemTime();

METHOD PRIVATE CalculateEfficiency : BOOL
VAR_IN_OUT
	powerstack 				: st_Powerstack_get;
	powermonitor			: st_powermonitor_get;
	system					: ST_system_get;
	battery					: ST_bms_get;
END_VAR

VAR_INST
	r_RawEfficiency	: REAL;
	r_AverageEfficiency: REAL;
	r_RoundtripEfficiency: REAL;
	
	
	ton_SumTimer			: TON :=(PT := T#100ms);
	r_EfficiencySum			: REAL;
	w_AverageSumCounter			: WORD;
END_VAR
r_RawEfficiency := ABS(powerstack.r_DCPower) / MAX(1,ABS(powermonitor.InputField.ar_ActivePower[0] + powermonitor.OutputField.ar_ActivePower[0])) * 100;

system.r_CurrentEfficiency := LIMIT(0, r_rawEfficiency, 99.8);

//manual averaging of the last hour of operation
ton_SumTimer(IN := NOT ton_SumTimer.Q);
IF powerstack.b_StartedState AND ton_SumTimer.Q THEN
	//reset counter and sum after 3000 samples +- 5min.
	IF w_AverageSumCounter = 3000 THEN
		//increment array index to add new efficiency value until upperbound has been reached.
		r_efficiencySum := r_efficiencySum - r_AverageEfficiency + system.r_CurrentEfficiency;
	ELSE
		//add new value to the summation
		w_AverageSumCounter := w_AverageSumCounter +1;
		r_EfficiencySum := r_efficiencySum + system.r_CurrentEfficiency;
	END_IF
	
	//System average efficiency during operation
	r_AverageEfficiency := r_EfficiencySum / MAX(1, w_AverageSumCounter);
	system.r_AvgEfficiency := r_AverageEfficiency;
	r_RoundtripEfficiency := LIMIT(0, powermonitor.BESS.r_EnergySupplied / MAX(1,powermonitor.BESS.r_EnergyConsumed - Battery.BatteryInfo.r_RemainingDischargeEnergyNett) * 100, 99);
	System.r_RoundtripEfficiency := r_RoundtripEfficiency;
END_IF
END_METHOD

METHOD ConfigureOutputContact : BOOL
VAR_INPUT
	SignalSelect			: eOutputContactSignal;
	GensetStartStop			: BOOL;
END_VAR
CASE SignalSelect OF
	eOutputContactSignal.FireAlarm 		: ConfigureOutputContact:= monitor.protections.FireDetection.b_FireAlarm;
	eOutputContactSignal.GenStartStop 	: ConfigureOutputContact:= GensetStartStop;
END_CASE
END_METHOD

METHOD EMstop : BOOL
VAR_INPUT
END_VAR

VAR_INST
	ton_FBdelay : TON := (PT:= T#20MS);
END_VAR
EMstop := FALSE;
ton_FBdelay(IN:= TRUE);

IF ton_FBdelay.Q THEN
	ton_FBdelay.IN := FALSE;
	EMstop := TRUE;
END_IF
END_METHOD

METHOD FillSystemMonitoringVars : BOOL

VAR_INST
	st_Params_MA			: ST_CTRL_MOVING_AVERAGE_PARAMS;
	ui_filterSize			: UINT := 50;
	fb_AverageEff			: FB_CTRL_MOVING_AVERAGE;
END_VAR
monitor.b_modeSwitchEnable := monitor.system.e_State = eSystemstate.Off OR 
	monitor.system.e_State = eSystemstate.StandBy OR
	monitor.system.e_State = eSystemstate.Init OR
	monitor.system.e_State = eSystemstate.Conditioning OR
	monitor.system.e_State = eSystemstate.Transport OR 
	monitor.system.e_State = eSystemstate.Dehumidifying OR
	monitor.system.e_State = eSystemState.EMstop; 

//Effiencies
monitor.system.b_StartAllowed := 
	control.HardSettings.system.e_EarthingSystem <> 0 AND
	monitor.powerstack.b_StartEnabled AND monitor.Cooling.ui_DehumRemainingTime = 0;
monitor.system.s_SystemName := Monitor.Router.Mobile.s_EmergencySMSDevName;

CASE toSystem.powerstack.e_Powermode OF
	ePowermodes.Droop: monitor.system.e_UgridPowermode := eUgridPowermode.Droop;
	ePowermodes.DroopZeroStart: monitor.system.e_UgridPowermode := eUgridPowermode.DroopZeroStart;
	ePowermodes.Isochronous: monitor.system.e_UgridPowermode := eUgridPowermode.Isochronous;
END_CASE

CASE toSystem.powerstack.e_InverterMode OF
	eInvertermodes.Afe : 
		monitor.system.e_gridmode := eGridmode.following;
		monitor.system.e_UgridPowermode := eUgridPowermode.None;
	eInvertermodes.Microgrid : monitor.system.e_gridmode := eGridmode.forming;
END_CASE
END_METHOD

METHOD GetDiagnostics
VAR_IN_OUT
	AddError		: ARRAY [*] OF FB_AddErrorST;
	a_ActiveEvents	: ARRAY [*] OF ST_ErrorStruct;
	w_Index			: WORD;
END_VAR
GenGridControl.GetDiagnostics(AddError, a_ActiveEvents, w_Index);
PowerControl.GetDiagnostics(AddError, a_ActiveEvents, w_Index);

(*Machine name update pending*) 	AddError[w_Index](
		b_ErrorTrig				:= monitor.system.events.b_RestartRequiredMachineName,
		out_ST_Error			:= a_ActiveEvents[w_Index],
		w_ErrorID				:= 1,
		e_ObjectID				:= eObject_ID.system,
		s_Message				:= 'Machinename update pending in VDL Powernet: System restart required',
		e_sev					:= eseverity.Info
		);
	w_Index := w_Index +1;
	
(*Machine name update pending*) AddError[w_Index](
		b_ErrorTrig				:= monitor.HartingIO.b_ExtSystemShutdownRequest,
		out_ST_Error			:= a_ActiveEvents[w_Index],
		w_ErrorID				:= 2,
		e_ObjectID				:= eObject_ID.system,
		s_Message				:= 'External IO initiated system shutdown',
		e_sev					:= eseverity.NormalShutdown,
		b_autoclear				:= FALSE
		);
	w_Index := w_Index +1;
	
(*time update failed*)	AddError[w_Index](
			b_ErrorTrig				:= monitor.system.events.b_TimeUpdateFailed,
			b_SMSEnableVDL			:= FALSE,
			out_ST_Error			:= a_ActiveEvents[w_Index],
			w_ErrorID				:= 3,					
			s_Message				:= 'System time update failed',
			e_sev					:= eSeverity.info,
			b_AutoClear				:= TRUE,
			e_ErrAckAccess			:= eErrAckAccess.General
			);
		w_Index := w_Index +1;
END_METHOD

METHOD GetEvents : BOOL
VAR_INPUT
END_VAR

VAR_INST
	s_machineNameOld : STRING;
	initdone		: BOOL;
END_VAR
IF NOT initdone AND monitor.system.s_SystemName <> '' THEN
	s_machineNameOld := monitor.system.s_SystemName;
	initdone := TRUE;
END_IF

monitor.system.events.b_RestartRequiredMachineName := s_machineNameOld <> monitor.system.s_SystemName;
END_METHOD

METHOD JsonFileToStruct : BOOL
VAR_INPUT
	bExecute			: BOOL;
	sJsonPathname		: STRING := 'C:\PLC_Utility\CalData_Powerstack.json';
	sStructName			: STRING;
	pStruct				: PVOID;
	nStruct				: UDINT;
	WriteMode			: BOOL;
	
END_VAR

VAR_OUTPUT
	Busy			: BOOL;
	Error			: BOOL;
	sMessage		: STRING;
END_VAR

VAR_INST
	bEnableCreateFile 	: BOOL := TRUE;
	SfcstepPrev		: BYTE;
	SFCTransAllowed	: BOOL;
	tofSFCstepDelay	: TOF := (PT := T#20MS);
	fbFileRead 		: FB_FileRead;
	fbFileWrite		: FB_FileWrite;
	fbFileOpen		: FB_FileOpen;
	fbFileClose		: FB_FileClose;
	sErrorMessage	: STRING;
	bLoading 		: BOOL;
	ton_executedelay	: TON := (PT := T#10MS);
	SFCstep			: BYTE;
	bLoad			: BOOL;
	bError			: BOOL;
	bfileOpened		: BOOL;
	hrErrorCode		: HRESULT;
	fbJson         : FB_JsonSaxWriter;
  	fbJsonDataType : FB_JsonReadWriteDataType;
  	sJsonDoc     	: STRING(10000);
	nBytesRead		: UDINT;
	b_CreateNewFile 	: BOOL;
	bOpenExecute		: BOOL;
	bReadExecute		: BOOL;
	bWriteExecute		: BOOL;
	bCloseExecute		: BOOL;
	nModeSel			: DWORD;	
	udLength			: UDINT;
	tDelayWriting		: TON := (PT := T#50MS);
	bEnable : BOOL := FALSE;
	
END_VAR
 

IF NOT ton_executedelay.Q THEN
	sfcstep := 0;
END_IF

IF pStruct = 0 THEN
	sfcstep := 99;
	sErrorMessage := 'Invalid pointer to struct';
ELSIF nStruct = 0 THEN
	sfcstep := 99;
	sErrorMessage := 'Invalid size of struct';
END_IF

//transition delay logic.
tofSFCstepDelay(IN := SFCstep <> SFCstepPrev);
SFCTransAllowed := NOT tofSFCstepDelay.Q AND bLoading;

CASE SFCstep OF
0: //idle
bEnable := FALSE;
	bLoading := FALSE;
	bError := FALSE;
	SFCTransAllowed := FALSE;
	bOpenExecute 			:= FALSE;
	bReadExecute 			:= FALSE;
	bWriteExecute 			:= FALSE;
	bCloseExecute 			:= FALSE;
	bEnableCreateFile 		:= FALSE;
	
	ton_executedelay(IN := bExecute);
	
	IF ton_executedelay.Q THEN
		sfcstep := SEL(writemode OR b_CreateNewFile, 1, 2);
		nModeSel 		:= SEL(sfcstep = 1, FOPEN_MODEWRITE,FOPEN_MODEREAD);
		sErrorMessage := '';
		bLoading := TRUE;	
	END_IF
	
1: 	//open file
	sJsonDoc := '';
	nModeSel 				:= FOPEN_MODEREAD;
	bReadExecute 			:= FALSE;
	bWriteExecute 			:= FALSE;
	bCloseExecute 			:= FALSE;
	bOpenExecute 			:= SFCTransAllowed;
	
	
	IF bEnable THEN 
	//IF SFCTransAllowed THEN
		IF fbFileOpen.hfile <> 0 AND NOT fbFileOpen.bBusy AND NOT fbFileOpen.bError THEN
			SFCstep := 10;
			bEnable := FALSE;
		ELSIF fbFileOpen.bError THEN
			sErrorMessage := CONCAT('Error opening file: sfc step ', TO_STRING(sfcstep));
			sfcstep := SEL(bEnableCreateFile, 97, 2);
		END_IF
	END_IF
	
2: //create file if non existing
	sJsonDoc := '';
	b_createNewFile := FALSE;
	nModeSel 				:= FOPEN_MODEWRITE;
	bReadExecute 			:= FALSE;
	bWriteExecute 			:= FALSE;
	bCloseExecute 			:= FALSE;
	bOpenExecute 			:= SFCTransAllowed;

	
	IF bEnable THEN 
		IF fbFileOpen.hfile <> 0 AND NOT fbFileOpen.bBusy AND NOT fbFileOpen.bError THEN
			sErrorMessage := 'New file created';
			sJsonDoc 		:= '';
			MEMSET(ADR(sJsonDoc), 0, SIZEOF(sJsonDoc));
			SFCstep := 3;
			bEnable := FALSE;
		ELSIF fbFileOpen.bError THEN
			sErrorMessage := CONCAT('Error opening and creating file: sfc step ', TO_STRING(sfcstep));
			sfcstep := 97;
		END_IF
	END_IF
	
3: //Write current struct values to new Json string
//	IF LEN(sJsonDoc) = 0 THEN
		fbJson.ResetDocument();
		fbJsonDataType.AddJsonValueFromSymbol(fbJson, sStructName, nStruct, pStruct, hrErrorCode => hrErrorCode);
		udLength := fbJson.GetDocumentLength();
		fbJson.CopyDocument(sJsonDoc, udLength);
//	END_IF
	
	IF SFCTransAllowed THEN
		IF hrErrorCode = 0 THEN
			bError := FALSE;
			sfcstep := 4; //final step
		ELSE
			bError := TRUE;
			sErrorMessage := CONCAT('Error generating json string: SFC step ', TO_STRING(sfcstep));
			sfcstep := 97; //error step
		END_IF
	END_IF
	
4: //write json string to file
	bReadExecute 	:= FALSE;
	bOpenExecute 	:= FALSE;
	bCloseExecute 	:= FALSE;
	bWriteExecute 	:= SFCTransAllowed;
	
	IF SFCTransAllowed THEN
		IF NOT fbFileWrite.bBusy AND NOT fbFileWrite.bError THEN
			SFCstep := 97;
			bEnable := FALSE;
		ELSIF fbFileWrite.bError THEN
			sErrorMessage := CONCAT('Error writing file: sfc step ', TO_STRING(sfcstep));
			sfcstep := 97;
		END_IF
	END_IF
		
10: //Read File
	sJsonDoc 		:= '';
	bOpenExecute 	:= FALSE;
	bWriteExecute 	:= FALSE;
	bCloseExecute 	:= FALSE;
	bReadExecute 	:= SFCTransAllowed;
	
	IF SFCTransAllowed THEN
		IF NOT fbFileRead.bBusy AND NOT fbFileRead.bError THEN
			SFCstep := 11;
			bEnable := FALSE;
		ELSIF fbFileRead.bError THEN
			sErrorMessage := CONCAT('Error reading file: sfc step ', TO_STRING(sfcstep));
			sfcstep :=  97;
			b_createNewFile := bEnableCreateFile;
		END_IF
	END_IF

	
11: //Convert buffer to struct
	fbJsonDataType.SetSymbolFromJson(sJsonDoc, sStructName, nStruct, pStruct, hrErrorCode => hrErrorCode);
	
	IF SFCTransAllowed THEN
		
		IF hrErrorCode = 0 THEN
			bError := FALSE;
			sfcstep := 97; //final step
		ELSE
			bError := TRUE;
			sErrorMessage := CONCAT('Error writing file to struct: sfc step ', TO_STRING(sfcstep));
			sfcstep := 97;
			b_createNewFile := bEnableCreateFile;	
		END_IF
	END_IF

97: // file opened
	
	bWriteExecute 	:= FALSE;
	bOpenExecute 	:= FALSE;
	bReadExecute 	:= FALSE;
	bCloseExecute 	:= bfileOpened := fbFileOpen.hFile <> 0;

	
	IF SFCTransAllowed THEN
		IF NOT fbFileClose.bBusy AND NOT fbFileClose.bError THEN
			bfileOpened := FALSE;
			sfcstep := 98;
			bEnable := FALSE;
		ELSIF fbFileClose.bError THEN
			sErrorMessage := CONCAT('Error closing file ', TO_STRING(sfcstep));
			bError := TRUE;
			sfcstep := 98;
		END_IF
	END_IF
	
98: 	//feedback and reset method for next request
	IF NOT bError THEN
		sErrorMessage := 'SUCCES';
	ELSE
		Error := TRUE;
	END_IF
	bEnable := FALSE;
	bOpenExecute 		:= FALSE;
	bReadExecute 		:= FALSE;
	bWriteExecute 		:= FALSE;
	bCloseExecute 		:= FALSE;
	ton_executedelay.IN := FALSE;
	sfcstep := 99;
	
	
99: //once here, reset SFC
	IF NOT b_CreateNewFile THEN
		JsonFileToStruct := TRUE;
	END_IF
	sfcstep := 0;
END_CASE
	


fbFileOpen(sPathName:= sJsonPathname , nMode := nModeSel ,bExecute:= bOpenExecute);
fbFileWrite(hFile := fbFileOpen.hFile , pWriteBuff := ADR(sJsonDoc),bExecute := bWriteExecute , cbWriteLen := udLength);
fbFileRead(hFile := fbFileOpen.hFile, pReadBuff := ADR(sJsonDoc), cbReadLen := SIZEOF(sJsonDoc),bExecute := bReadExecute, cbRead => nBytesRead);
fbFileClose(hFile := fbFileOpen.hFile, bExecute := bCloseExecute);

IF fbFileOpen.bBusy AND bOpenExecute THEN
	bOpenExecute := FALSE;
	bEnable := TRUE;
END_IF
//	rTrigExecute(CLK := FALSE);
//	IF NOT rTrigExecute.CLK THEN
//		JsonFileToStruct := TRUE;
SFCstepPrev := SFCstep;

//output data
busy := bLoading;
sMessage := sErrorMessage;
END_METHOD

METHOD MapUsercontrolsToSystemVars : BOOL

VAR_INST
	FrequencySetpoint : REAL;
	VoltageSetpoint : REAL;
	rs_ACDCChargerEnable	: RS;
	
END_VAR
VAR_INST // added by the converter: edge detectors and wires of the graphical bodies
    _rt1, _rt2, _rt3 : R_TRIG;
    _w1, _w2 : BOOL;
END_VAR
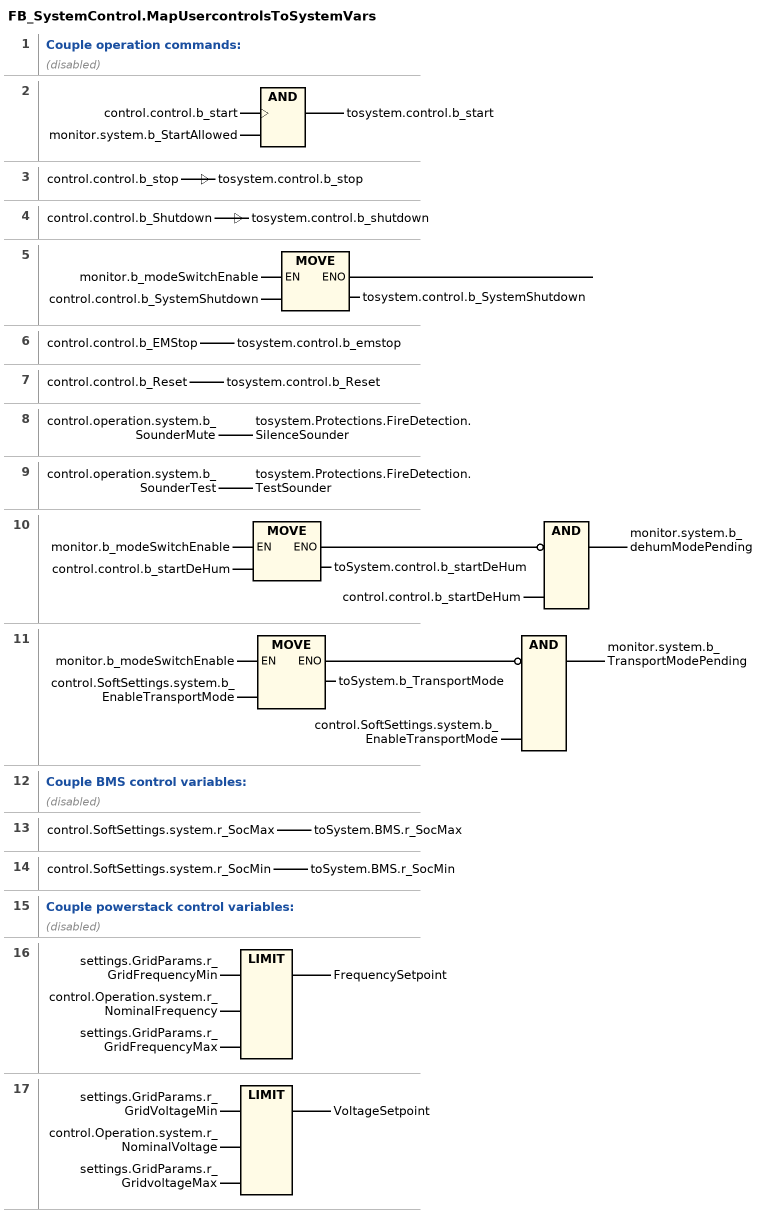
// NETWORK 1 (disabled)
// label: Couple operation commands

// NETWORK 2
_rt1(CLK := control.control.b_start);
tosystem.control.b_start := _rt1.Q AND monitor.system.b_StartAllowed;

// NETWORK 3
_rt2(CLK := control.control.b_stop);
tosystem.control.b_stop := _rt2.Q;

// NETWORK 4
_rt3(CLK := control.control.b_Shutdown);
tosystem.control.b_shutdown := _rt3.Q;

// NETWORK 5
IF monitor.b_modeSwitchEnable THEN tosystem.control.b_SystemShutdown := control.control.b_SystemShutdown; END_IF

// NETWORK 6
tosystem.control.b_emstop := control.control.b_EMStop;

// NETWORK 7
tosystem.control.b_Reset := control.control.b_Reset;

// NETWORK 8
tosystem.Protections.FireDetection.SilenceSounder := control.operation.system.b_SounderMute;

// NETWORK 9
tosystem.Protections.FireDetection.TestSounder := control.operation.system.b_SounderTest;

// NETWORK 10
_w1 := monitor.b_modeSwitchEnable;
IF _w1 THEN toSystem.control.b_startDeHum := control.control.b_startDeHum; END_IF
monitor.system.b_dehumModePending := NOT _w1 AND control.control.b_startDeHum;

// NETWORK 11
_w2 := monitor.b_modeSwitchEnable;
IF _w2 THEN toSystem.b_TransportMode := control.SoftSettings.system.b_EnableTransportMode; END_IF
monitor.system.b_TransportModePending := NOT _w2 AND control.SoftSettings.system.b_EnableTransportMode;

// NETWORK 12 (disabled)
// label: Couple BMS control variables

// NETWORK 13
toSystem.BMS.r_SocMax := control.SoftSettings.system.r_SocMax;

// NETWORK 14
toSystem.BMS.r_SocMin := control.SoftSettings.system.r_SocMin;

// NETWORK 15 (disabled)
// label: Couple powerstack control variables

// NETWORK 16
FrequencySetpoint := LIMIT(settings.GridParams.r_GridFrequencyMin, control.Operation.system.r_NominalFrequency, settings.GridParams.r_GridFrequencyMax);

// NETWORK 17
VoltageSetpoint := LIMIT(settings.GridParams.r_GridVoltageMin, control.Operation.system.r_NominalVoltage, settings.GridParams.r_GridvoltageMax);

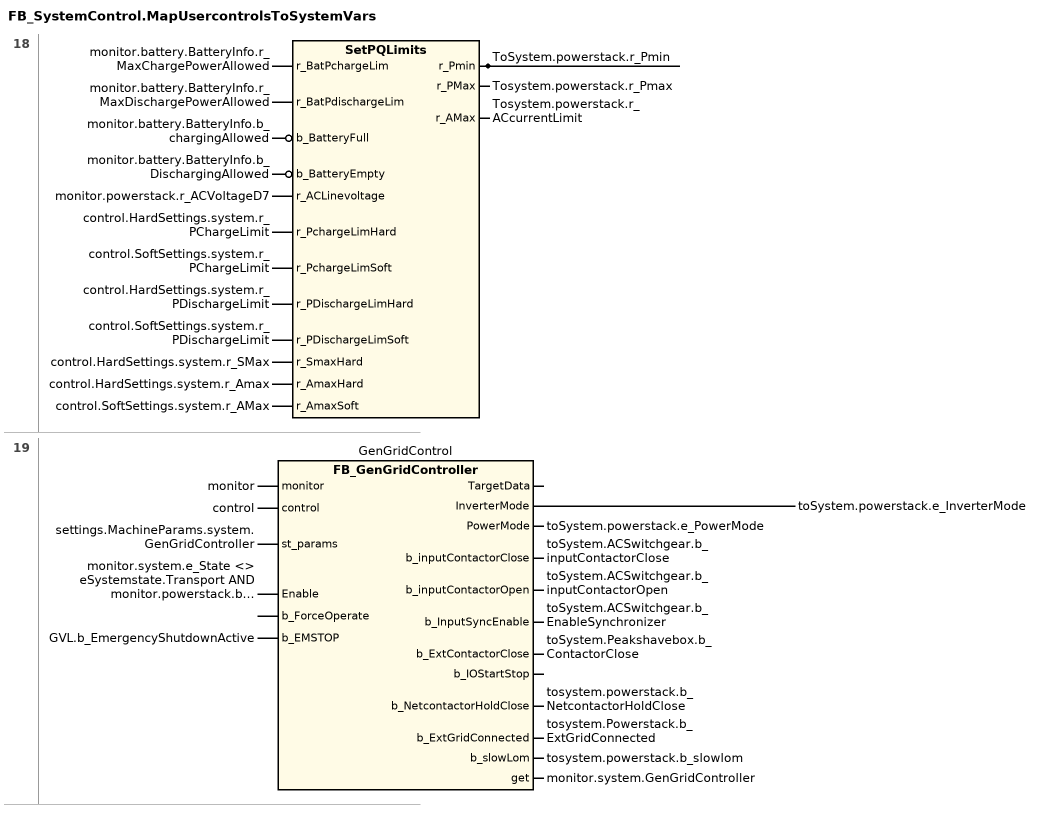
// NETWORK 18
SetPQLimits(r_BatPchargeLim := monitor.battery.BatteryInfo.r_MaxChargePowerAllowed, r_BatPdischargeLim := monitor.battery.BatteryInfo.r_MaxDischargePowerAllowed, b_BatteryFull := NOT monitor.battery.BatteryInfo.b_chargingAllowed, b_BatteryEmpty := NOT monitor.battery.BatteryInfo.b_DischargingAllowed, r_ACLinevoltage := monitor.powerstack.r_ACVoltageD7, r_PchargeLimHard := control.HardSettings.system.r_PChargeLimit, r_PchargeLimSoft := control.SoftSettings.system.r_PChargeLimit, r_PDischargeLimHard := control.HardSettings.system.r_PDischargeLimit, r_PDischargeLimSoft := control.SoftSettings.system.r_PDischargeLimit, r_SmaxHard := control.HardSettings.system.r_SMax, r_AmaxHard := control.HardSettings.system.r_Amax, r_AmaxSoft := control.SoftSettings.system.r_AMax, r_Pmin => ToSystem.powerstack.r_Pmin, r_PMax => Tosystem.powerstack.r_Pmax, r_AMax => Tosystem.powerstack.r_ACcurrentLimit);

// NETWORK 19
GenGridControl(
    monitor := monitor,
    control := control,
    st_params := settings.MachineParams.system.GenGridController,
    Enable := monitor.system.e_State <> eSystemstate.Transport AND monitor.powerstack.b_ControlEnabled,
    b_EMSTOP := GVL.b_EmergencyShutdownActive,
    PowerMode => toSystem.powerstack.e_PowerMode,
    b_inputContactorClose => toSystem.ACSwitchgear.b_inputContactorClose,
    b_inputContactorOpen => toSystem.ACSwitchgear.b_inputContactorOpen,
    b_InputSyncEnable => toSystem.ACSwitchgear.b_EnableSynchronizer,
    b_ExtContactorClose => toSystem.Peakshavebox.b_ContactorClose,
    b_NetcontactorHoldClose => tosystem.powerstack.b_NetcontactorHoldClose,
    b_ExtGridConnected => tosystem.Powerstack.b_ExtGridConnected,
    b_slowLom => tosystem.powerstack.b_slowlom,
    get => monitor.system.GenGridController); // FB_GenGridController
toSystem.powerstack.e_InverterMode := GenGridControl.InverterMode;

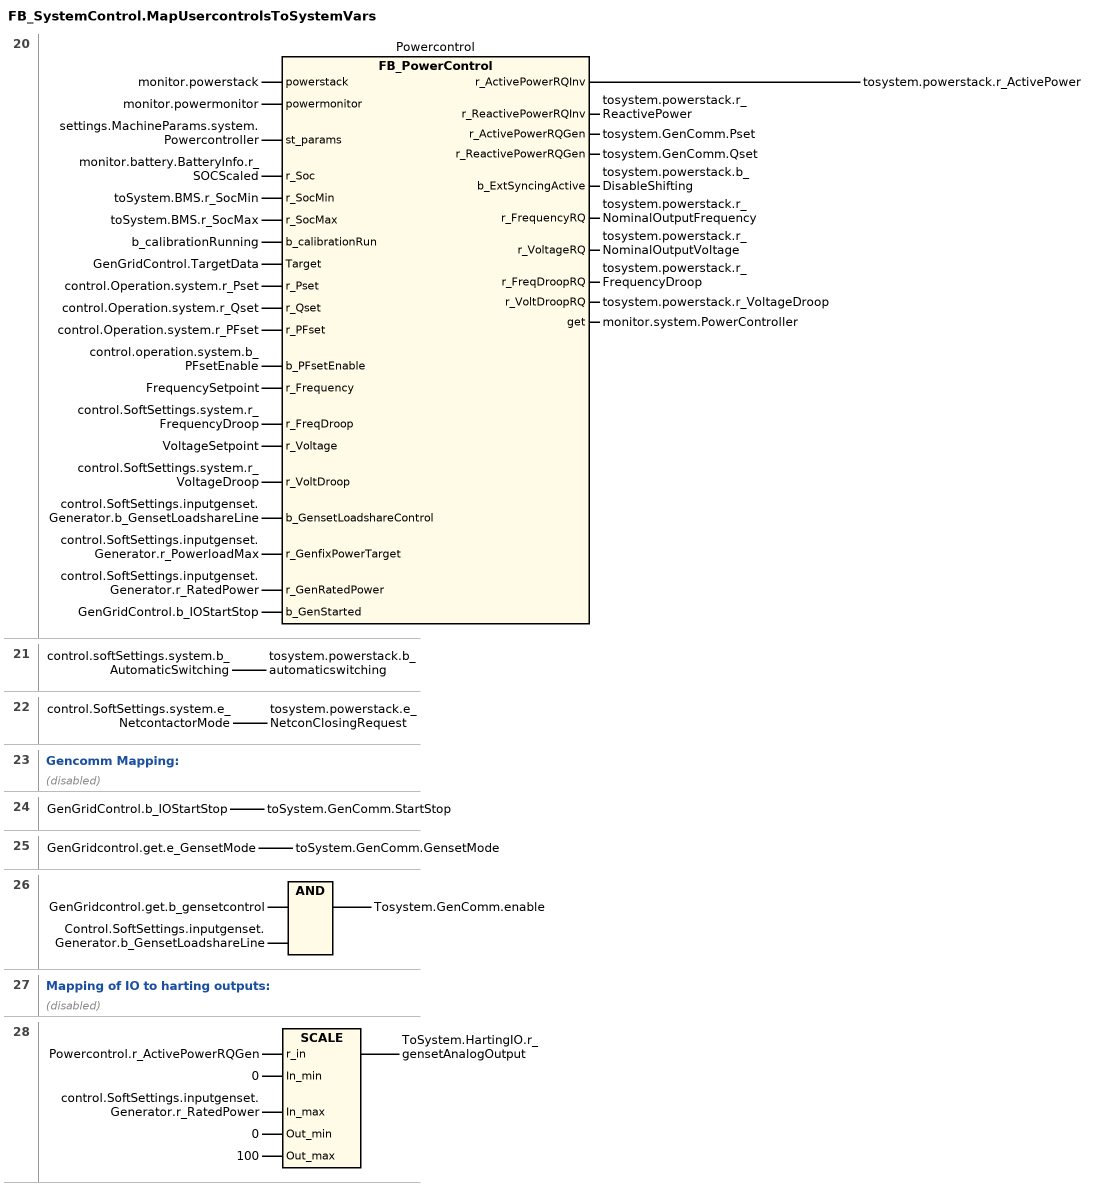
// NETWORK 20
Powercontrol(
    powerstack := monitor.powerstack,
    powermonitor := monitor.powermonitor,
    st_params := settings.MachineParams.system.Powercontroller,
    r_Soc := monitor.battery.BatteryInfo.r_SOCScaled,
    r_SocMin := toSystem.BMS.r_SocMin,
    r_SocMax := toSystem.BMS.r_SocMax,
    b_calibrationRun := b_calibrationRunning,
    Target := GenGridControl.TargetData,
    r_Pset := control.Operation.system.r_Pset,
    r_Qset := control.Operation.system.r_Qset,
    r_PFset := control.Operation.system.r_PFset,
    b_PFsetEnable := control.operation.system.b_PFsetEnable,
    r_Frequency := FrequencySetpoint,
    r_FreqDroop := control.SoftSettings.system.r_FrequencyDroop,
    r_Voltage := VoltageSetpoint,
    r_VoltDroop := control.SoftSettings.system.r_VoltageDroop,
    b_GensetLoadshareControl := control.SoftSettings.inputgenset.Generator.b_GensetLoadshareLine,
    r_GenfixPowerTarget := control.SoftSettings.inputgenset.Generator.r_PowerloadMax,
    r_GenRatedPower := control.SoftSettings.inputgenset.Generator.r_RatedPower,
    b_GenStarted := GenGridControl.b_IOStartStop,
    r_ReactivePowerRQInv => tosystem.powerstack.r_ReactivePower,
    r_ActivePowerRQGen => tosystem.GenComm.Pset,
    r_ReactivePowerRQGen => tosystem.GenComm.Qset,
    b_ExtSyncingActive => tosystem.powerstack.b_DisableShifting,
    r_FrequencyRQ => tosystem.powerstack.r_NominalOutputFrequency,
    r_VoltageRQ => tosystem.powerstack.r_NominalOutputVoltage,
    r_FreqDroopRQ => tosystem.powerstack.r_FrequencyDroop,
    r_VoltDroopRQ => tosystem.powerstack.r_VoltageDroop,
    get => monitor.system.PowerController); // FB_PowerControl
tosystem.powerstack.r_ActivePower := Powercontrol.r_ActivePowerRQInv;

// NETWORK 21
tosystem.powerstack.b_automaticswitching := control.softSettings.system.b_AutomaticSwitching;

// NETWORK 22
tosystem.powerstack.e_NetconClosingRequest := control.SoftSettings.system.e_NetcontactorMode;

// NETWORK 23 (disabled)
// label: Gencomm Mapping

// NETWORK 24
toSystem.GenComm.StartStop := GenGridControl.b_IOStartStop;

// NETWORK 25
toSystem.GenComm.GensetMode := GenGridcontrol.get.e_GensetMode;

// NETWORK 26
Tosystem.GenComm.enable := GenGridcontrol.get.b_gensetcontrol AND Control.SoftSettings.inputgenset.Generator.b_GensetLoadshareLine;

// NETWORK 27 (disabled)
// label: Mapping of IO to harting outputs

// NETWORK 28
ToSystem.HartingIO.r_gensetAnalogOutput := SCALE(r_in := Powercontrol.r_ActivePowerRQGen, In_min := 0, In_max := control.SoftSettings.inputgenset.Generator.r_RatedPower, Out_min := 0, Out_max := 100);

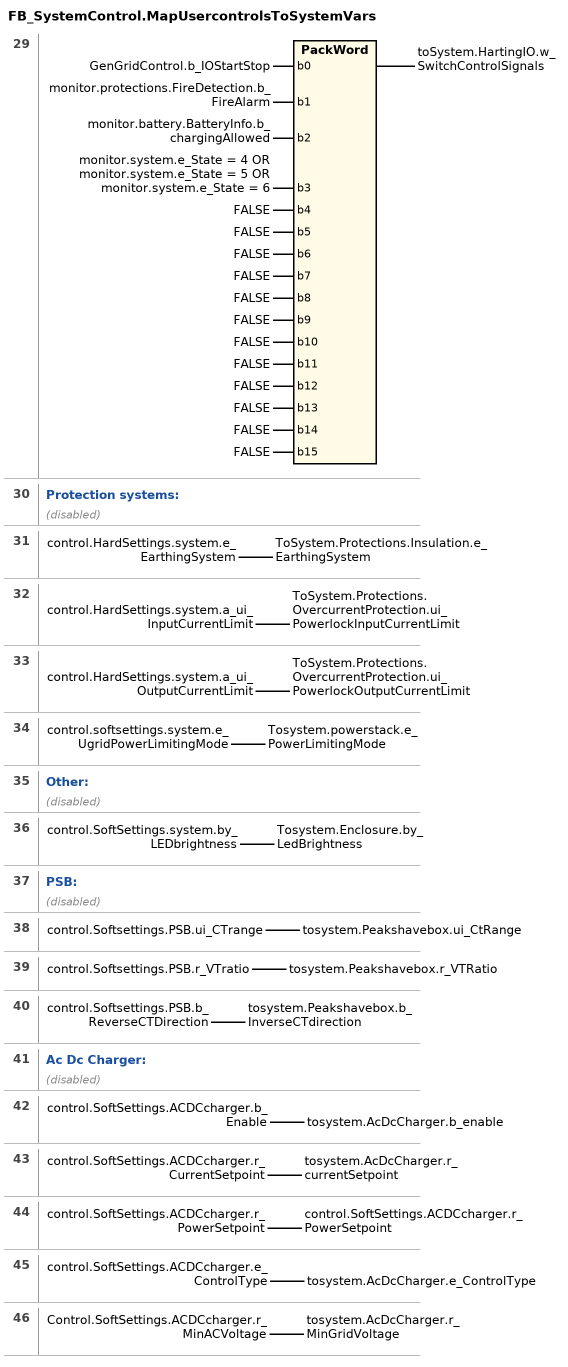
// NETWORK 29
toSystem.HartingIO.w_SwitchControlSignals := PackWord(b0 := GenGridControl.b_IOStartStop, b1 := monitor.protections.FireDetection.b_FireAlarm, b2 := monitor.battery.BatteryInfo.b_chargingAllowed, b3 := monitor.system.e_State = 4 OR monitor.system.e_State = 5 OR monitor.system.e_State = 6, b4 := FALSE, b5 := FALSE, b6 := FALSE, b7 := FALSE, b8 := FALSE, b9 := FALSE, b10 := FALSE, b11 := FALSE, b12 := FALSE, b13 := FALSE, b14 := FALSE, b15 := FALSE);

// NETWORK 30 (disabled)
// label: Protection systems

// NETWORK 31
ToSystem.Protections.Insulation.e_EarthingSystem := control.HardSettings.system.e_EarthingSystem;

// NETWORK 32
ToSystem.Protections.OvercurrentProtection.ui_PowerlockInputCurrentLimit := control.HardSettings.system.a_ui_InputCurrentLimit;

// NETWORK 33
ToSystem.Protections.OvercurrentProtection.ui_PowerlockOutputCurrentLimit := control.HardSettings.system.a_ui_OutputCurrentLimit;

// NETWORK 34
Tosystem.powerstack.e_PowerLimitingMode := control.softsettings.system.e_UgridPowerLimitingMode;

// NETWORK 35 (disabled)
// label: Other

// NETWORK 36
Tosystem.Enclosure.by_LedBrightness := control.SoftSettings.system.by_LEDbrightness;

// NETWORK 37 (disabled)
// label: PSB

// NETWORK 38
tosystem.Peakshavebox.ui_CtRange := control.Softsettings.PSB.ui_CTrange;

// NETWORK 39
tosystem.Peakshavebox.r_VTRatio := control.Softsettings.PSB.r_VTratio;

